LIN {X 0,Y 573.271,Z 613.194,A -85,B 0,C 180,E1 -2290.528,E2 -2290.528} C_VEL
LIN {X 0,Y 573.246,Z 613.204,A -85,B 0,C 180,E1 -2293.669,E2 -2293.669} C_VEL
LIN {X 0,Y 573.242,Z 613.198,A -85,B 0,C 180,E1 -2296.641,E2 -2296.641} C_VEL
LIN {X 0,Y 573.276,Z 613.202,A -85,B 0,C 180,E1 -2299.478,E2 -2299.478} C_VEL
LIN {X 0,Y 573.238,Z 613.198,A -85,B 0,C 180,E1 -2302.193,E2 -2302.193} C_VEL
LIN {X 0,Y 573.271,Z 613.195,A -85,B 0,C 180,E1 -2304.817,E2 -2304.817} C_VEL
LIN {X 0,Y 573.259,Z 613.2,A -85,B 0,C 180,E1 -2307.355,E2 -2307.355} C_VEL
LIN {X 0,Y 573.252,Z 613.206,A -85,B 0,C 180,E1 -2309.824,E2 -2309.824} C_VEL
LIN {X 0,Y 573.291,Z 613.195,A -85,B 0,C 180,E1 -2312.235,E2 -2312.235} C_VEL
LIN {X 0,Y 573.277,Z 613.196,A -85,B 0,C 180,E1 -2315.366,E2 -2315.366} C_VEL
LIN {X 0,Y 573.232,Z 613.202,A -85,B 0,C 180,E1 -2318.42,E2 -2318.42} C_VEL
LIN {X 0,Y 573.281,Z 613.193,A -85,B 0,C 180,E1 -2320.728,E2 -2320.728} C_VEL
LIN {X 0,Y 573.261,Z 613.2,A -85,B 0,C 180,E1 -2323.622,E2 -2323.622} C_VEL
LIN {X 0,Y 573.275,Z 613.2,A -85,B 0,C 180,E1 -2325.807,E2 -2325.807} C_VEL
LIN {X 0,Y 573.265,Z 613.197,A -85,B 0,C 180,E1 -2328.745,E2 -2328.745} C_VEL
LIN {X 0,Y 573.287,Z 613.193,A -85,B 0,C 180,E1 -2331.541,E2 -2331.541} C_VEL
LIN {X 0,Y 573.287,Z 613.2,A -85,B 0,C 180,E1 -2334.372,E2 -2334.372} C_VEL
LIN {X 0,Y 573.309,Z 613.19,A -85,B 0,C 180,E1 -2337.19,E2 -2337.19} C_VEL
LIN {X 0,Y 573.324,Z 613.193,A -85,B 0,C 180,E1 -2340,E2 -2340} C_VEL
LIN {X 0,Y 573.303,Z 613.194,A -85,B 0,C 180,E1 -2342.811,E2 -2342.811} C_VEL
LIN {X 0,Y 573.293,Z 613.191,A -85,B 0,C 180,E1 -2345.628,E2 -2345.628} C_VEL
LIN {X 0,Y 573.286,Z 613.203,A -85,B 0,C 180,E1 -2348.46,E2 -2348.46} C_VEL
LIN {X 0,Y 573.275,Z 613.194,A -85,B 0,C 180,E1 -2351.312,E2 -2351.312} C_VEL
LIN {X 0,Y 573.284,Z 613.2,A -85,B 0,C 180,E1 -2354.424,E2 -2354.424} C_VEL
LIN {X 0,Y 573.261,Z 613.199,A -85,B 0,C 180,E1 -2357.112,E2 -2357.112} C_VEL
LIN {X 0,Y 573.244,Z 613.198,A -85,B 0,C 180,E1 -2360.077,E2 -2360.077} C_VEL
LIN {X 0,Y 573.234,Z 613.203,A -85,B 0,C 180,E1 -2362.338,E2 -2362.338} C_VEL
LIN {X 0,Y 573.248,Z 613.2,A -85,B 0,C 180,E1 -2364.387,E2 -2364.387} C_VEL
LIN {X 0,Y 572.619,Z 613.286,A -85,B 0,C 180,E1 -2364.973,E2 -2364.973} C_VEL
LIN {X 0,Y 569.76,Z 613.642,A -85,B 0,C 180,E1 -2365.924,E2 -2365.924} C_VEL
LIN {X 0,Y 567.315,Z 613.945,A -85,B 0,C 180,E1 -2366.689,E2 -2366.689} C_VEL
LIN {X 0,Y 566.258,Z 614.07,A -85,B 0,C 180,E1 -2367.281,E2 -2367.281} C_VEL
LIN {X 0,Y 566.17,Z 614.079,A -85,B 0,C 180,E1 -2367.481,E2 -2367.481} C_VEL
LIN {X 0,Y 566.199,Z 614.073,A -85,B 0,C 180,E1 -2369.769,E2 -2369.769} C_VEL
LIN {X 0,Y 566.206,Z 614.077,A -85,B 0,C 180,E1 -2372.43,E2 -2372.43} C_VEL
LIN {X 0,Y 566.18,Z 614.088,A -85,B 0,C 180,E1 -2374.989,E2 -2374.989} C_VEL
LIN {X 0,Y 566.197,Z 614.08,A -85,B 0,C 180,E1 -2377.461,E2 -2377.461} C_VEL
LIN {X 0,Y 566.209,Z 614.073,A -85,B 0,C 180,E1 -2380.199,E2 -2380.199} C_VEL
LIN {X 0,Y 566.184,Z 614.087,A -85,B 0,C 180,E1 -2383.056,E2 -2383.056} C_VEL
LIN {X 0,Y 566.159,Z 614.081,A -85,B 0,C 180,E1 -2386.053,E2 -2386.053} C_VEL
LIN {X 0,Y 566.167,Z 614.084,A -85,B 0,C 180,E1 -2388.86,E2 -2388.86} C_VEL
LIN {X 0,Y 566.206,Z 614.084,A -85,B 0,C 180,E1 -2391.443,E2 -2391.443} C_VEL
LIN {X 0,Y 566.148,Z 614.082,A -85,B 0,C 180,E1 -2394.307,E2 -2394.307} C_VEL
LIN {X 0,Y 566.198,Z 614.078,A -85,B 0,C 180,E1 -2396.896,E2 -2396.896} C_VEL
LIN {X 0,Y 566.169,Z 614.089,A -85,B 0,C 180,E1 -2399.407,E2 -2399.407} C_VEL
LIN {X 0,Y 566.174,Z 614.086,A -85,B 0,C 180,E1 -2401.855,E2 -2401.855} C_VEL
LIN {X 0,Y 566.21,Z 614.214,A -85,B 0,C 180,E1 -2404.103,E2 -2404.103} C_VEL
LIN {X 0,Y 566.783,Z 618.685,A -85,B 0,C 180,E1 -2404.849,E2 -2404.849} C_VEL
LIN {X 0,Y 566.52,Z 638.155,A -85,B 0,C 180,E1 -2407.959,E2 -2407.959} C_VEL
LIN {X 0,Y 566.539,Z 638.91,A -85,B 0,C 180,E1 -2408.08,E2 -2408.08} C_VEL
LIN {X 0,Y 567.797,Z 645.92,A -85,B 0,C 180,E1 -2408.214,E2 -2408.214} C_VEL
LIN {X 0,Y 567.426,Z 775.387,A -85,B 0,C 180,E1 -2409.89,E2 -2409.89} C_VEL
LIN {X 0,Y 567.273,Z 789.85,A -85,B 0,C 180,E1 -2410.224,E2 -2410.224} C_VEL
LIN {X 0,Y 567.158,Z 803.531,A -85,B 0,C 180,E1 -2410.689,E2 -2410.689} C_VEL
LIN {X 0,Y 566.982,Z 816.893,A -85,B 0,C 180,E1 -2411.293,E2 -2411.293} C_VEL
LIN {X 0,Y 566.77,Z 829.75,A -85,B 0,C 180,E1 -2412.034,E2 -2412.034} C_VEL
LIN {X 0,Y 566.592,Z 841.641,A -85,B 0,C 180,E1 -2412.884,E2 -2412.884} C_VEL
LIN {X 0,Y 566.402,Z 852.078,A -85,B 0,C 180,E1 -2413.789,E2 -2413.789} C_VEL
LIN {X 0,Y 566.259,Z 862.634,A -85,B 0,C 180,E1 -2414.892,E2 -2414.892} C_VEL
LIN {X 0,Y 566.111,Z 871.296,A -85,B 0,C 180,E1 -2415.991,E2 -2415.991} C_VEL
LIN {X 0,Y 566.028,Z 879.528,A -85,B 0,C 180,E1 -2417.268,E2 -2417.268} C_VEL
LIN {X 0,Y 565.938,Z 886.128,A -85,B 0,C 180,E1 -2418.539,E2 -2418.539} C_VEL
LIN {X 0,Y 565.917,Z 890.69,A -85,B 0,C 180,E1 -2419.626,E2 -2419.626} C_VEL
LIN {X 0,Y 565.877,Z 894.258,A -85,B 0,C 180,E1 -2420.709,E2 -2420.709} C_VEL
LIN {X 0,Y 565.882,Z 897.734,A -85,B 0,C 180,E1 -2422.148,E2 -2422.148} C_VEL
LIN {X 0,Y 565.899,Z 899.79,A -85,B 0,C 180,E1 -2423.583,E2 -2423.583} C_VEL
LIN {X 0,Y 565.844,Z 900.498,A -85,B 0,C 180,E1 -2425.012,E2 -2425.012} C_VEL
LIN {X 0,Y 565.885,Z 899.863,A -85,B 0,C 180,E1 -2426.44,E2 -2426.44} C_VEL
LIN {X 0,Y 565.839,Z 897.888,A -85,B 0,C 180,E1 -2427.865,E2 -2427.865} C_VEL
LIN {X 0,Y 565.848,Z 894.533,A -85,B 0,C 180,E1 -2429.288,E2 -2429.288} C_VEL
LIN {X 0,Y 565.89,Z 889.709,A -85,B 0,C 180,E1 -2430.712,E2 -2430.712} C_VEL
LIN {X 0,Y 566.002,Z 885.069,A -85,B 0,C 180,E1 -2431.779,E2 -2431.779} C_VEL
LIN {X 0,Y 566.061,Z 878.343,A -85,B 0,C 180,E1 -2433.025,E2 -2433.025} C_VEL
LIN {X 0,Y 566.16,Z 870.011,A -85,B 0,C 180,E1 -2434.271,E2 -2434.271} C_VEL
LIN {X 0,Y 566.241,Z 861.352,A -85,B 0,C 180,E1 -2435.341,E2 -2435.341} C_VEL
LIN {X 0,Y 566.433,Z 850.893,A -85,B 0,C 180,E1 -2436.412,E2 -2436.412} C_VEL
LIN {X 0,Y 566.652,Z 839.212,A -85,B 0,C 180,E1 -2437.393,E2 -2437.393} C_VEL
LIN {X 0,Y 566.807,Z 827.519,A -85,B 0,C 180,E1 -2438.198,E2 -2438.198} C_VEL
LIN {X 0,Y 566.977,Z 814.646,A -85,B 0,C 180,E1 -2438.914,E2 -2438.914} C_VEL
LIN {X 0,Y 567.184,Z 801.171,A -85,B 0,C 180,E1 -2439.495,E2 -2439.495} C_VEL
LIN {X 0,Y 567.297,Z 787.032,A -85,B 0,C 180,E1 -2439.943,E2 -2439.943} C_VEL
LIN {X 0,Y 567.415,Z 773.297,A -85,B 0,C 180,E1 -2440.234,E2 -2440.234} C_VEL
LIN {X 0,Y 567.787,Z 645.918,A -85,B 0,C 180,E1 -2441.877,E2 -2441.877} C_VEL
LIN {X 0,Y 566.495,Z 638.792,A -85,B 0,C 180,E1 -2442.03,E2 -2442.03} C_VEL
LIN {X 0,Y 566.712,Z 622.116,A -85,B 0,C 180,E1 -2444.69,E2 -2444.69} C_VEL
LIN {X 0,Y 566.544,Z 616.194,A -85,B 0,C 180,E1 -2445.653,E2 -2445.653} C_VEL
LIN {X 0,Y 566.179,Z 614.087,A -85,B 0,C 180,E1 -2446.033,E2 -2446.033} C_VEL
LIN {X 0,Y 566.172,Z 614.088,A -85,B 0,C 180,E1 -2448.829,E2 -2448.829} C_VEL
LIN {X 0,Y 566.211,Z 614.076,A -85,B 0,C 180,E1 -2451.419,E2 -2451.419} C_VEL
LIN {X 0,Y 566.154,Z 614.085,A -85,B 0,C 180,E1 -2454.183,E2 -2454.183} C_VEL
LIN {X 0,Y 566.165,Z 614.09,A -85,B 0,C 180,E1 -2456.649,E2 -2456.649} C_VEL
LIN {X 0,Y 566.159,Z 614.081,A -85,B 0,C 180,E1 -2459.771,E2 -2459.771} C_VEL
LIN {X 0,Y 566.18,Z 614.082,A -85,B 0,C 180,E1 -2462.425,E2 -2462.425} C_VEL
LIN {X 0,Y 566.165,Z 614.089,A -85,B 0,C 180,E1 -2464.986,E2 -2464.986} C_VEL
LIN {X 0,Y 566.188,Z 614.079,A -85,B 0,C 180,E1 -2467.462,E2 -2467.462} C_VEL
LIN {X 0,Y 566.169,Z 614.077,A -85,B 0,C 180,E1 -2470.203,E2 -2470.203} C_VEL
LIN {X 0,Y 566.181,Z 614.087,A -85,B 0,C 180,E1 -2473.056,E2 -2473.056} C_VEL
LIN {X 0,Y 566.158,Z 614.081,A -85,B 0,C 180,E1 -2476.053,E2 -2476.053} C_VEL
LIN {X 0,Y 566.154,Z 614.087,A -85,B 0,C 180,E1 -2478.858,E2 -2478.858} C_VEL
LIN {X 0,Y 566.201,Z 614.078,A -85,B 0,C 180,E1 -2481.444,E2 -2481.444} C_VEL
LIN {X 0,Y 566.145,Z 614.08,A -85,B 0,C 180,E1 -2484.306,E2 -2484.306} C_VEL
LIN {X 0,Y 566.2,Z 614.08,A -85,B 0,C 180,E1 -2486.896,E2 -2486.896} C_VEL
LIN {X 0,Y 566.171,Z 614.086,A -85,B 0,C 180,E1 -2489.406,E2 -2489.406} C_VEL
LIN {X 0,Y 566.191,Z 614.079,A -85,B 0,C 180,E1 -2491.856,E2 -2491.856} C_VEL
LIN {X 0,Y 566.185,Z 614.077,A -85,B 0,C 180,E1 -2494.249,E2 -2494.249} C_VEL
LIN {X 0,Y 566.169,Z 614.078,A -85,B 0,C 180,E1 -2496.72,E2 -2496.72} C_VEL
LIN {X 0,Y 566.208,Z 614.081,A -85,B 0,C 180,E1 -2499.662,E2 -2499.662} C_VEL
LIN {X 0,Y 566.197,Z 614.073,A -85,B 0,C 180,E1 -2502.668,E2 -2502.668} C_VEL
LIN {X 0,Y 566.237,Z 614.08,A -85,B 0,C 180,E1 -2505.627,E2 -2505.627} C_VEL
LIN {X 0,Y 566.239,Z 614.069,A -85,B 0,C 180,E1 -2508.675,E2 -2508.675} C_VEL
LIN {X 0,Y 566.226,Z 614.077,A -85,B 0,C 180,E1 -2511.434,E2 -2511.434} C_VEL
LIN {X 0,Y 566.25,Z 614.07,A -85,B 0,C 180,E1 -2514.301,E2 -2514.301} C_VEL
LIN {X 0,Y 566.283,Z 614.074,A -85,B 0,C 180,E1 -2517.866,E2 -2517.866} C_VEL
LIN {X 0,Y 566.302,Z 614.062,A -85,B 0,C 180,E1 -2520.711,E2 -2520.711} C_VEL
LIN {X 0,Y 566.273,Z 614.066,A -85,B 0,C 180,E1 -2522.845,E2 -2522.845} C_VEL
LIN {X 0,Y 566.256,Z 614.075,A -85,B 0,C 180,E1 -2525.698,E2 -2525.698} C_VEL
LIN {X 0,Y 566.23,Z 614.073,A -85,B 0,C 180,E1 -2528.566,E2 -2528.566} C_VEL
LIN {X 0,Y 566.245,Z 614.071,A -85,B 0,C 180,E1 -2531.454,E2 -2531.454} C_VEL
LIN {X 0,Y 566.238,Z 614.073,A -85,B 0,C 180,E1 -2534.506,E2 -2534.506} C_VEL
LIN {X 0,Y 566.203,Z 614.075,A -85,B 0,C 180,E1 -2537.331,E2 -2537.331} C_VEL
LIN {X 0,Y 566.217,Z 614.08,A -85,B 0,C 180,E1 -2540.337,E2 -2540.337} C_VEL
LIN {X 0,Y 566.172,Z 614.078,A -85,B 0,C 180,E1 -2543.281,E2 -2543.281} C_VEL
LIN {X 0,Y 566.215,Z 614.076,A -85,B 0,C 180,E1 -2545.749,E2 -2545.749} C_VEL
LIN {X 0,Y 566.205,Z 614.084,A -85,B 0,C 180,E1 -2548.202,E2 -2548.202} C_VEL
LIN {X 0,Y 566.197,Z 614.076,A -85,B 0,C 180,E1 -2551.077,E2 -2551.077} C_VEL
LIN {X 0,Y 566.215,Z 614.075,A -85,B 0,C 180,E1 -2553.734,E2 -2553.734} C_VEL
LIN {X 0,Y 566.203,Z 614.083,A -85,B 0,C 180,E1 -2556.57,E2 -2556.57} C_VEL
LIN {X 0,Y 566.224,Z 614.072,A -85,B 0,C 180,E1 -2559.273,E2 -2559.273} C_VEL
LIN {X 0,Y 566.194,Z 614.08,A -85,B 0,C 180,E1 -2562.089,E2 -2562.089} C_VEL
LIN {X 0,Y 566.175,Z 614.081,A -85,B 0,C 180,E1 -2565.036,E2 -2565.036} C_VEL
LIN {X 0,Y 566.221,Z 614.076,A -85,B 0,C 180,E1 -2568.136,E2 -2568.136} C_VEL
LIN {X 0,Y 566.218,Z 614.083,A -85,B 0,C 180,E1 -2570.726,E2 -2570.726} C_VEL
LIN {X 0,Y 566.22,Z 614.074,A -85,B 0,C 180,E1 -2573.783,E2 -2573.783} C_VEL
LIN {X 0,Y 566.215,Z 614.077,A -85,B 0,C 180,E1 -2576.266,E2 -2576.266} C_VEL
LIN {X 0,Y 566.202,Z 614.084,A -85,B 0,C 180,E1 -2578.922,E2 -2578.922} C_VEL
LIN {X 0,Y 566.214,Z 614.075,A -85,B 0,C 180,E1 -2581.857,E2 -2581.857} C_VEL
LIN {X 0,Y 566.22,Z 614.081,A -85,B 0,C 180,E1 -2584.644,E2 -2584.644} C_VEL
LIN {X 0,Y 566.24,Z 614.207,A -85,B 0,C 180,E1 -2584.792,E2 -2584.792} C_VEL
LIN {X 0,Y 567.536,Z 620.359,A -85,B 0,C 180,E1 -2585.685,E2 -2585.685} C_VEL
LIN {X 0,Y 567.212,Z 640.232,A -85,B 0,C 180,E1 -2588.323,E2 -2588.323} C_VEL
LIN {X 0,Y 566.892,Z 662.255,A -85,B 0,C 180,E1 -2591.196,E2 -2591.196} C_VEL
LIN {X 0,Y 566.687,Z 676.414,A -85,B 0,C 180,E1 -2593.018,E2 -2593.018} C_VEL
LIN {X 0,Y 567.814,Z 683.83,A -85,B 0,C 180,E1 -2593.155,E2 -2593.155} C_VEL
LIN {X 0,Y 567.43,Z 814.879,A -85,B 0,C 180,E1 -2594.855,E2 -2594.855} C_VEL
LIN {X 0,Y 567.273,Z 829.536,A -85,B 0,C 180,E1 -2595.2,E2 -2595.2} C_VEL
LIN {X 0,Y 567.102,Z 843.837,A -85,B 0,C 180,E1 -2595.695,E2 -2595.695} C_VEL
LIN {X 0,Y 566.964,Z 856.64,A -85,B 0,C 180,E1 -2596.286,E2 -2596.286} C_VEL
LIN {X 0,Y 566.787,Z 869.098,A -85,B 0,C 180,E1 -2597.012,E2 -2597.012} C_VEL
LIN {X 0,Y 566.576,Z 880.478,A -85,B 0,C 180,E1 -2597.826,E2 -2597.826} C_VEL
LIN {X 0,Y 566.452,Z 891.045,A -85,B 0,C 180,E1 -2598.742,E2 -2598.742} C_VEL
LIN {X 0,Y 566.247,Z 901.333,A -85,B 0,C 180,E1 -2599.813,E2 -2599.813} C_VEL
LIN {X 0,Y 566.153,Z 909.911,A -85,B 0,C 180,E1 -2600.893,E2 -2600.893} C_VEL
LIN {X 0,Y 566.059,Z 918.115,A -85,B 0,C 180,E1 -2602.15,E2 -2602.15} C_VEL
LIN {X 0,Y 565.966,Z 924.801,A -85,B 0,C 180,E1 -2603.422,E2 -2603.422} C_VEL
LIN {X 0,Y 565.927,Z 929.961,A -85,B 0,C 180,E1 -2604.656,E2 -2604.656} C_VEL
LIN {X 0,Y 565.957,Z 933.443,A -85,B 0,C 180,E1 -2605.727,E2 -2605.727} C_VEL
LIN {X 0,Y 565.874,Z 936.831,A -85,B 0,C 180,E1 -2607.152,E2 -2607.152} C_VEL
LIN {X 0,Y 565.84,Z 938.832,A -85,B 0,C 180,E1 -2608.576,E2 -2608.576} C_VEL
LIN {X 0,Y 565.837,Z 939.5,A -85,B 0,C 180,E1 -2610,E2 -2610} C_VEL
LIN {X 0,Y 565.84,Z 938.833,A -85,B 0,C 180,E1 -2611.423,E2 -2611.423} C_VEL
LIN {X 0,Y 565.874,Z 936.833,A -85,B 0,C 180,E1 -2612.847,E2 -2612.847} C_VEL
LIN {X 0,Y 565.956,Z 933.445,A -85,B 0,C 180,E1 -2614.273,E2 -2614.273} C_VEL
LIN {X 0,Y 565.988,Z 928.568,A -85,B 0,C 180,E1 -2615.701,E2 -2615.701} C_VEL
LIN {X 0,Y 565.992,Z 924.045,A -85,B 0,C 180,E1 -2616.739,E2 -2616.739} C_VEL
LIN {X 0,Y 566.047,Z 917.038,A -85,B 0,C 180,E1 -2618.029,E2 -2618.029} C_VEL
LIN {X 0,Y 566.177,Z 908.559,A -85,B 0,C 180,E1 -2619.286,E2 -2619.286} C_VEL
LIN {X 0,Y 566.294,Z 899.708,A -85,B 0,C 180,E1 -2620.367,E2 -2620.367} C_VEL
LIN {X 0,Y 566.485,Z 888.991,A -85,B 0,C 180,E1 -2621.449,E2 -2621.449} C_VEL
LIN {X 0,Y 566.629,Z 878.143,A -85,B 0,C 180,E1 -2622.354,E2 -2622.354} C_VEL
LIN {X 0,Y 566.8,Z 866.259,A -85,B 0,C 180,E1 -2623.17,E2 -2623.17} C_VEL
LIN {X 0,Y 567.02,Z 853.096,A -85,B 0,C 180,E1 -2623.895,E2 -2623.895} C_VEL
LIN {X 0,Y 567.192,Z 840.055,A -85,B 0,C 180,E1 -2624.453,E2 -2624.453} C_VEL
LIN {X 0,Y 567.324,Z 826.235,A -85,B 0,C 180,E1 -2624.892,E2 -2624.892} C_VEL
LIN {X 0,Y 567.455,Z 812.133,A -85,B 0,C 180,E1 -2625.19,E2 -2625.19} C_VEL
LIN {X 0,Y 567.765,Z 682.287,A -85,B 0,C 180,E1 -2626.867,E2 -2626.867} C_VEL
LIN {X 0,Y 566.685,Z 676.417,A -85,B 0,C 180,E1 -2626.981,E2 -2626.981} C_VEL
LIN {X 0,Y 566.979,Z 655.178,A -85,B 0,C 180,E1 -2629.723,E2 -2629.723} C_VEL
LIN {X 0,Y 567.374,Z 631.917,A -85,B 0,C 180,E1 -2632.774,E2 -2632.774} C_VEL
LIN {X 0,Y 567.535,Z 620.36,A -85,B 0,C 180,E1 -2634.315,E2 -2634.315} C_VEL
LIN {X 0,Y 566.224,Z 614.081,A -85,B 0,C 180,E1 -2635.257,E2 -2635.257} C_VEL
LIN {X 0,Y 566.231,Z 614.074,A -85,B 0,C 180,E1 -2638.142,E2 -2638.142} C_VEL
LIN {X 0,Y 566.201,Z 614.084,A -85,B 0,C 180,E1 -2641.078,E2 -2641.078} C_VEL
LIN {X 0,Y 566.214,Z 614.077,A -85,B 0,C 180,E1 -2643.734,E2 -2643.734} C_VEL
LIN {X 0,Y 566.218,Z 614.074,A -85,B 0,C 180,E1 -2646.569,E2 -2646.569} C_VEL
LIN {X 0,Y 566.214,Z 614.078,A -85,B 0,C 180,E1 -2649.686,E2 -2649.686} C_VEL
LIN {X 0,Y 566.215,Z 614.075,A -85,B 0,C 180,E1 -2652.087,E2 -2652.087} C_VEL
LIN {X 0,Y 566.174,Z 614.081,A -85,B 0,C 180,E1 -2655.036,E2 -2655.036} C_VEL
LIN {X 0,Y 566.22,Z 614.074,A -85,B 0,C 180,E1 -2658.136,E2 -2658.136} C_VEL
LIN {X 0,Y 566.224,Z 614.073,A -85,B 0,C 180,E1 -2660.727,E2 -2660.727} C_VEL
LIN {X 0,Y 566.22,Z 614.081,A -85,B 0,C 180,E1 -2663.783,E2 -2663.783} C_VEL
LIN {X 0,Y 566.214,Z 614.075,A -85,B 0,C 180,E1 -2666.266,E2 -2666.266} C_VEL
LIN {X 0,Y 566.201,Z 614.071,A -85,B 0,C 180,E1 -2668.922,E2 -2668.922} C_VEL
LIN {X 0,Y 566.231,Z 614.081,A -85,B 0,C 180,E1 -2671.858,E2 -2671.858} C_VEL
LIN {X 0,Y 566.215,Z 614.077,A -85,B 0,C 180,E1 -2674.251,E2 -2674.251} C_VEL
LIN {X 0,Y 566.193,Z 614.076,A -85,B 0,C 180,E1 -2676.714,E2 -2676.714} C_VEL
LIN {X 0,Y 566.216,Z 614.079,A -85,B 0,C 180,E1 -2679.663,E2 -2679.663} C_VEL
LIN {X 0,Y 566.206,Z 614.076,A -85,B 0,C 180,E1 -2682.669,E2 -2682.669} C_VEL
LIN {X 0,Y 566.236,Z 614.074,A -85,B 0,C 180,E1 -2685.627,E2 -2685.627} C_VEL
LIN {X 0,Y 566.237,Z 614.073,A -85,B 0,C 180,E1 -2688.675,E2 -2688.675} C_VEL
LIN {X 0,Y 566.23,Z 614.071,A -85,B 0,C 180,E1 -2691.434,E2 -2691.434} C_VEL
LIN {X 0,Y 566.256,Z 614.077,A -85,B 0,C 180,E1 -2694.302,E2 -2694.302} C_VEL
LIN {X 0,Y 566.282,Z 614.069,A -85,B 0,C 180,E1 -2697.866,E2 -2697.866} C_VEL
LIN {X 0,Y 566.3,Z 614.067,A -85,B 0,C 180,E1 -2700.711,E2 -2700.711} C_VEL
LIN {X 0,Y 566.27,Z 614.07,A -85,B 0,C 180,E1 -2702.846,E2 -2702.846} C_VEL
LIN {X 0,Y 566.262,Z 614.067,A -85,B 0,C 180,E1 -2705.698,E2 -2705.698} C_VEL
LIN {X 0,Y 566.229,Z 614.081,A -85,B 0,C 180,E1 -2708.566,E2 -2708.566} C_VEL
LIN {X 0,Y 566.245,Z 614.07,A -85,B 0,C 180,E1 -2711.455,E2 -2711.455} C_VEL
LIN {X 0,Y 566.237,Z 614.08,A -85,B 0,C 180,E1 -2714.507,E2 -2714.507} C_VEL
LIN {X 0,Y 566.201,Z 614.077,A -85,B 0,C 180,E1 -2717.332,E2 -2717.332} C_VEL
LIN {X 0,Y 566.21,Z 614.077,A -85,B 0,C 180,E1 -2720.338,E2 -2720.338} C_VEL
LIN {X 0,Y 566.17,Z 614.081,A -85,B 0,C 180,E1 -2723.281,E2 -2723.281} C_VEL
LIN {X 0,Y 566.206,Z 614.075,A -85,B 0,C 180,E1 -2725.75,E2 -2725.75} C_VEL
LIN {X 0,Y 566.17,Z 614.079,A -85,B 0,C 180,E1 -2727.481,E2 -2727.481} C_VEL
LIN {X 0,Y 565.499,Z 614.162,A -85,B 0,C 180,E1 -2728.075,E2 -2728.075} C_VEL
LIN {X 0,Y 562.646,Z 614.523,A -85,B 0,C 180,E1 -2729.039,E2 -2729.039} C_VEL
LIN {X 0,Y 560.242,Z 614.818,A -85,B 0,C 180,E1 -2729.815,E2 -2729.815} C_VEL
LIN {X 0,Y 559.217,Z 614.945,A -85,B 0,C 180,E1 -2730.414,E2 -2730.414} C_VEL
LIN {X 0,Y 559.137,Z 614.957,A -85,B 0,C 180,E1 -2730.616,E2 -2730.616} C_VEL
LIN {X 0,Y 559.154,Z 614.96,A -85,B 0,C 180,E1 -2732.716,E2 -2732.716} C_VEL
LIN {X 0,Y 559.129,Z 614.961,A -85,B 0,C 180,E1 -2735.324,E2 -2735.324} C_VEL
LIN {X 0,Y 559.131,Z 614.956,A -85,B 0,C 180,E1 -2738.018,E2 -2738.018} C_VEL
LIN {X 0,Y 559.155,Z 614.957,A -85,B 0,C 180,E1 -2740.813,E2 -2740.813} C_VEL
LIN {X 0,Y 559.111,Z 614.961,A -85,B 0,C 180,E1 -2743.737,E2 -2743.737} C_VEL
LIN {X 0,Y 559.11,Z 614.959,A -85,B 0,C 180,E1 -2746.263,E2 -2746.263} C_VEL
LIN {X 0,Y 559.155,Z 614.963,A -85,B 0,C 180,E1 -2749.187,E2 -2749.187} C_VEL
LIN {X 0,Y 559.131,Z 614.958,A -85,B 0,C 180,E1 -2751.982,E2 -2751.982} C_VEL
LIN {X 0,Y 559.127,Z 614.958,A -85,B 0,C 180,E1 -2754.789,E2 -2754.789} C_VEL
LIN {X 0,Y 559.152,Z 614.96,A -85,B 0,C 180,E1 -2757.366,E2 -2757.366} C_VEL
LIN {X 0,Y 559.12,Z 614.96,A -85,B 0,C 180,E1 -2760.149,E2 -2760.149} C_VEL
LIN {X 0,Y 559.114,Z 614.967,A -85,B 0,C 180,E1 -2763.185,E2 -2763.185} C_VEL
LIN {X 0,Y 559.163,Z 614.979,A -85,B 0,C 180,E1 -2763.952,E2 -2763.952} C_VEL
LIN {X 0,Y 559.795,Z 619.574,A -85,B 0,C 180,E1 -2764.732,E2 -2764.732} C_VEL
LIN {X 0,Y 559.524,Z 637.72,A -85,B 0,C 180,E1 -2767.669,E2 -2767.669} C_VEL
LIN {X 0,Y 559.518,Z 638.927,A -85,B 0,C 180,E1 -2767.863,E2 -2767.863} C_VEL
LIN {X 0,Y 561.012,Z 646.832,A -85,B 0,C 180,E1 -2768.016,E2 -2768.016} C_VEL
LIN {X 0,Y 560.608,Z 774.759,A -85,B 0,C 180,E1 -2769.69,E2 -2769.69} C_VEL
LIN {X 0,Y 560.462,Z 788.934,A -85,B 0,C 180,E1 -2770.012,E2 -2770.012} C_VEL
LIN {X 0,Y 560.274,Z 803.153,A -85,B 0,C 180,E1 -2770.493,E2 -2770.493} C_VEL
LIN {X 0,Y 560.077,Z 815.624,A -85,B 0,C 180,E1 -2771.053,E2 -2771.053} C_VEL
LIN {X 0,Y 559.86,Z 827.273,A -85,B 0,C 180,E1 -2771.71,E2 -2771.71} C_VEL
LIN {X 0,Y 559.653,Z 839.346,A -85,B 0,C 180,E1 -2772.55,E2 -2772.55} C_VEL
LIN {X 0,Y 559.469,Z 849.397,A -85,B 0,C 180,E1 -2773.394,E2 -2773.394} C_VEL
LIN {X 0,Y 559.287,Z 858.744,A -85,B 0,C 180,E1 -2774.326,E2 -2774.326} C_VEL
LIN {X 0,Y 559.123,Z 868.85,A -85,B 0,C 180,E1 -2775.545,E2 -2775.545} C_VEL
LIN {X 0,Y 558.994,Z 876.943,A -85,B 0,C 180,E1 -2776.735,E2 -2776.735} C_VEL
LIN {X 0,Y 558.888,Z 884.071,A -85,B 0,C 180,E1 -2778.025,E2 -2778.025} C_VEL
LIN {X 0,Y 558.859,Z 889.002,A -85,B 0,C 180,E1 -2779.127,E2 -2779.127} C_VEL
LIN {X 0,Y 558.793,Z 894.072,A -85,B 0,C 180,E1 -2780.59,E2 -2780.59} C_VEL
LIN {X 0,Y 558.801,Z 897.609,A -85,B 0,C 180,E1 -2782.048,E2 -2782.048} C_VEL
LIN {X 0,Y 558.827,Z 899.723,A -85,B 0,C 180,E1 -2783.501,E2 -2783.501} C_VEL
LIN {X 0,Y 558.759,Z 900.485,A -85,B 0,C 180,E1 -2784.949,E2 -2784.949} C_VEL
LIN {X 0,Y 558.797,Z 899.919,A -85,B 0,C 180,E1 -2786.395,E2 -2786.395} C_VEL
LIN {X 0,Y 558.744,Z 898.012,A -85,B 0,C 180,E1 -2787.838,E2 -2787.838} C_VEL
LIN {X 0,Y 558.749,Z 894.718,A -85,B 0,C 180,E1 -2789.279,E2 -2789.279} C_VEL
LIN {X 0,Y 558.796,Z 889.957,A -85,B 0,C 180,E1 -2790.721,E2 -2790.721} C_VEL
LIN {X 0,Y 558.91,Z 885.373,A -85,B 0,C 180,E1 -2791.802,E2 -2791.802} C_VEL
LIN {X 0,Y 559.008,Z 878.725,A -85,B 0,C 180,E1 -2793.063,E2 -2793.063} C_VEL
LIN {X 0,Y 559.12,Z 870.481,A -85,B 0,C 180,E1 -2794.325,E2 -2794.325} C_VEL
LIN {X 0,Y 559.21,Z 861.916,A -85,B 0,C 180,E1 -2795.409,E2 -2795.409} C_VEL
LIN {X 0,Y 559.411,Z 851.567,A -85,B 0,C 180,E1 -2796.492,E2 -2796.492} C_VEL
LIN {X 0,Y 559.659,Z 840.024,A -85,B 0,C 180,E1 -2797.486,E2 -2797.486} C_VEL
LIN {X 0,Y 559.857,Z 828.502,A -85,B 0,C 180,E1 -2798.3,E2 -2798.3} C_VEL
LIN {X 0,Y 560.043,Z 815.863,A -85,B 0,C 180,E1 -2799.025,E2 -2799.025} C_VEL
LIN {X 0,Y 560.291,Z 802.768,A -85,B 0,C 180,E1 -2799.613,E2 -2799.613} C_VEL
LIN {X 0,Y 560.472,Z 788.582,A -85,B 0,C 180,E1 -2800.088,E2 -2800.088} C_VEL
LIN {X 0,Y 560.571,Z 774.462,A -85,B 0,C 180,E1 -2800.406,E2 -2800.406} C_VEL
LIN {X 0,Y 560.974,Z 646.407,A -85,B 0,C 180,E1 -2802.081,E2 -2802.081} C_VEL
LIN {X 0,Y 559.505,Z 638.834,A -85,B 0,C 180,E1 -2802.243,E2 -2802.243} C_VEL
LIN {X 0,Y 559.794,Z 621.074,A -85,B 0,C 180,E1 -2805.113,E2 -2805.113} C_VEL
LIN {X 0,Y 559.465,Z 616.617,A -85,B 0,C 180,E1 -2805.856,E2 -2805.856} C_VEL
LIN {X 0,Y 559.136,Z 614.965,A -85,B 0,C 180,E1 -2806.147,E2 -2806.147} C_VEL
LIN {X 0,Y 559.139,Z 614.961,A -85,B 0,C 180,E1 -2809.075,E2 -2809.075} C_VEL
LIN {X 0,Y 559.155,Z 614.955,A -85,B 0,C 180,E1 -2811.548,E2 -2811.548} C_VEL
LIN {X 0,Y 559.092,Z 614.969,A -85,B 0,C 180,E1 -2814.508,E2 -2814.508} C_VEL
LIN {X 0,Y 559.112,Z 614.967,A -85,B 0,C 180,E1 -2816.905,E2 -2816.905} C_VEL
LIN {X 0,Y 559.109,Z 614.959,A -85,B 0,C 180,E1 -2819.849,E2 -2819.849} C_VEL
LIN {X 0,Y 559.138,Z 614.964,A -85,B 0,C 180,E1 -2822.717,E2 -2822.717} C_VEL
LIN {X 0,Y 559.117,Z 614.961,A -85,B 0,C 180,E1 -2825.325,E2 -2825.325} C_VEL
LIN {X 0,Y 559.125,Z 614.957,A -85,B 0,C 180,E1 -2828.018,E2 -2828.018} C_VEL
LIN {X 0,Y 559.105,Z 614.964,A -85,B 0,C 180,E1 -2830.817,E2 -2830.817} C_VEL
LIN {X 0,Y 559.11,Z 614.959,A -85,B 0,C 180,E1 -2833.737,E2 -2833.737} C_VEL
LIN {X 0,Y 559.109,Z 614.959,A -85,B 0,C 180,E1 -2836.262,E2 -2836.262} C_VEL
LIN {X 0,Y 559.127,Z 614.966,A -85,B 0,C 180,E1 -2839.185,E2 -2839.185} C_VEL
LIN {X 0,Y 559.124,Z 614.953,A -85,B 0,C 180,E1 -2841.981,E2 -2841.981} C_VEL
LIN {X 0,Y 559.127,Z 614.958,A -85,B 0,C 180,E1 -2844.788,E2 -2844.788} C_VEL
LIN {X 0,Y 559.156,Z 614.961,A -85,B 0,C 180,E1 -2847.365,E2 -2847.365} C_VEL
LIN {X 0,Y 559.121,Z 614.956,A -85,B 0,C 180,E1 -2850.148,E2 -2850.148} C_VEL
LIN {X 0,Y 559.127,Z 614.957,A -85,B 0,C 180,E1 -2852.285,E2 -2852.285} C_VEL
LIN {X 0,Y 559.141,Z 614.956,A -85,B 0,C 180,E1 -2854.822,E2 -2854.822} C_VEL
LIN {X 0,Y 559.142,Z 614.958,A -85,B 0,C 180,E1 -2857.847,E2 -2857.847} C_VEL
LIN {X 0,Y 559.196,Z 614.947,A -85,B 0,C 180,E1 -2860.494,E2 -2860.494} C_VEL
LIN {X 0,Y 559.18,Z 614.952,A -85,B 0,C 180,E1 -2863.197,E2 -2863.197} C_VEL
LIN {X 0,Y 559.17,Z 614.953,A -85,B 0,C 180,E1 -2866.184,E2 -2866.184} C_VEL
LIN {X 0,Y 559.196,Z 614.949,A -85,B 0,C 180,E1 -2869.133,E2 -2869.133} C_VEL
LIN {X 0,Y 559.201,Z 614.951,A -85,B 0,C 180,E1 -2872.053,E2 -2872.053} C_VEL
LIN {X 0,Y 559.245,Z 614.942,A -85,B 0,C 180,E1 -2874.953,E2 -2874.953} C_VEL
LIN {X 0,Y 559.255,Z 614.95,A -85,B 0,C 180,E1 -2877.839,E2 -2877.839} C_VEL
LIN {X 0,Y 559.273,Z 614.937,A -85,B 0,C 180,E1 -2880.72,E2 -2880.72} C_VEL
LIN {X 0,Y 559.239,Z 614.943,A -85,B 0,C 180,E1 -2882.881,E2 -2882.881} C_VEL
LIN {X 0,Y 559.225,Z 614.952,A -85,B 0,C 180,E1 -2885.77,E2 -2885.77} C_VEL
LIN {X 0,Y 559.189,Z 614.95,A -85,B 0,C 180,E1 -2888.674,E2 -2888.674} C_VEL
LIN {X 0,Y 559.208,Z 614.949,A -85,B 0,C 180,E1 -2891.6,E2 -2891.6} C_VEL
LIN {X 0,Y 559.204,Z 614.948,A -85,B 0,C 180,E1 -2894.595,E2 -2894.595} C_VEL
LIN {X 0,Y 559.162,Z 614.954,A -85,B 0,C 180,E1 -2897.557,E2 -2897.557} C_VEL
LIN {X 0,Y 559.176,Z 614.955,A -85,B 0,C 180,E1 -2899.837,E2 -2899.837} C_VEL
LIN {X 0,Y 559.144,Z 614.965,A -85,B 0,C 180,E1 -2902.153,E2 -2902.153} C_VEL
LIN {X 0,Y 559.179,Z 614.95,A -85,B 0,C 180,E1 -2905.298,E2 -2905.298} C_VEL
LIN {X 0,Y 559.16,Z 614.954,A -85,B 0,C 180,E1 -2907.713,E2 -2907.713} C_VEL
LIN {X 0,Y 559.157,Z 614.961,A -85,B 0,C 180,E1 -2910.182,E2 -2910.182} C_VEL
LIN {X 0,Y 559.178,Z 614.954,A -85,B 0,C 180,E1 -2912.714,E2 -2912.714} C_VEL
LIN {X 0,Y 559.133,Z 614.956,A -85,B 0,C 180,E1 -2915.324,E2 -2915.324} C_VEL
LIN {X 0,Y 559.137,Z 614.959,A -85,B 0,C 180,E1 -2918.017,E2 -2918.017} C_VEL
LIN {X 0,Y 559.177,Z 614.955,A -85,B 0,C 180,E1 -2920.811,E2 -2920.811} C_VEL
LIN {X 0,Y 559.144,Z 614.955,A -85,B 0,C 180,E1 -2923.734,E2 -2923.734} C_VEL
LIN {X 0,Y 559.167,Z 614.958,A -85,B 0,C 180,E1 -2926.801,E2 -2926.801} C_VEL
LIN {X 0,Y 559.18,Z 614.952,A -85,B 0,C 180,E1 -2929.189,E2 -2929.189} C_VEL
LIN {X 0,Y 559.136,Z 614.957,A -85,B 0,C 180,E1 -2931.982,E2 -2931.982} C_VEL
LIN {X 0,Y 559.163,Z 614.962,A -85,B 0,C 180,E1 -2934.783,E2 -2934.783} C_VEL
LIN {X 0,Y 559.177,Z 614.953,A -85,B 0,C 180,E1 -2937.361,E2 -2937.361} C_VEL
LIN {X 0,Y 559.152,Z 614.956,A -85,B 0,C 180,E1 -2940.142,E2 -2940.142} C_VEL
LIN {X 0,Y 559.185,Z 614.958,A -85,B 0,C 180,E1 -2943.17,E2 -2943.17} C_VEL
LIN {X 0,Y 559.221,Z 615.119,A -85,B 0,C 180,E1 -2944.579,E2 -2944.579} C_VEL
LIN {X 0,Y 560.643,Z 621.803,A -85,B 0,C 180,E1 -2945.564,E2 -2945.564} C_VEL
LIN {X 0,Y 560.374,Z 639.14,A -85,B 0,C 180,E1 -2947.898,E2 -2947.898} C_VEL
LIN {X 0,Y 559.983,Z 659.702,A -85,B 0,C 180,E1 -2950.618,E2 -2950.618} C_VEL
LIN {X 0,Y 559.762,Z 676.392,A -85,B 0,C 180,E1 -2952.799,E2 -2952.799} C_VEL
LIN {X 0,Y 561.019,Z 684.077,A -85,B 0,C 180,E1 -2952.948,E2 -2952.948} C_VEL
LIN {X 0,Y 560.581,Z 814.879,A -85,B 0,C 180,E1 -2954.665,E2 -2954.665} C_VEL
LIN {X 0,Y 560.405,Z 829.139,A -85,B 0,C 180,E1 -2955.002,E2 -2955.002} C_VEL
LIN {X 0,Y 560.247,Z 842.707,A -85,B 0,C 180,E1 -2955.47,E2 -2955.47} C_VEL
LIN {X 0,Y 560.055,Z 856.641,A -85,B 0,C 180,E1 -2956.114,E2 -2956.114} C_VEL
LIN {X 0,Y 559.841,Z 869.099,A -85,B 0,C 180,E1 -2956.848,E2 -2956.848} C_VEL
LIN {X 0,Y 559.617,Z 880.479,A -85,B 0,C 180,E1 -2957.673,E2 -2957.673} C_VEL
LIN {X 0,Y 559.454,Z 891.643,A -85,B 0,C 180,E1 -2958.655,E2 -2958.655} C_VEL
LIN {X 0,Y 559.239,Z 901.332,A -85,B 0,C 180,E1 -2959.684,E2 -2959.684} C_VEL
LIN {X 0,Y 559.114,Z 909.911,A -85,B 0,C 180,E1 -2960.778,E2 -2960.778} C_VEL
LIN {X 0,Y 558.979,Z 918.115,A -85,B 0,C 180,E1 -2962.05,E2 -2962.05} C_VEL
LIN {X 0,Y 558.894,Z 925.165,A -85,B 0,C 180,E1 -2963.42,E2 -2963.42} C_VEL
LIN {X 0,Y 558.858,Z 929.961,A -85,B 0,C 180,E1 -2964.588,E2 -2964.588} C_VEL
LIN {X 0,Y 558.866,Z 933.443,A -85,B 0,C 180,E1 -2965.673,E2 -2965.673} C_VEL
LIN {X 0,Y 558.796,Z 936.832,A -85,B 0,C 180,E1 -2967.116,E2 -2967.116} C_VEL
LIN {X 0,Y 558.74,Z 938.833,A -85,B 0,C 180,E1 -2968.558,E2 -2968.558} C_VEL
LIN {X 0,Y 558.738,Z 939.5,A -85,B 0,C 180,E1 -2970,E2 -2970} C_VEL
LIN {X 0,Y 558.74,Z 938.834,A -85,B 0,C 180,E1 -2971.441,E2 -2971.441} C_VEL
LIN {X 0,Y 558.795,Z 936.834,A -85,B 0,C 180,E1 -2972.884,E2 -2972.884} C_VEL
LIN {X 0,Y 558.866,Z 933.445,A -85,B 0,C 180,E1 -2974.327,E2 -2974.327} C_VEL
LIN {X 0,Y 558.917,Z 928.568,A -85,B 0,C 180,E1 -2975.773,E2 -2975.773} C_VEL
LIN {X 0,Y 558.907,Z 922.053,A -85,B 0,C 180,E1 -2977.224,E2 -2977.224} C_VEL
LIN {X 0,Y 559.028,Z 914.801,A -85,B 0,C 180,E1 -2978.495,E2 -2978.495} C_VEL
LIN {X 0,Y 559.146,Z 905.823,A -85,B 0,C 180,E1 -2979.769,E2 -2979.769} C_VEL
LIN {X 0,Y 559.35,Z 896.392,A -85,B 0,C 180,E1 -2980.863,E2 -2980.863} C_VEL
LIN {X 0,Y 559.521,Z 885.951,A -85,B 0,C 180,E1 -2981.869,E2 -2981.869} C_VEL
LIN {X 0,Y 559.715,Z 874.435,A -85,B 0,C 180,E1 -2982.786,E2 -2982.786} C_VEL
LIN {X 0,Y 559.951,Z 861.645,A -85,B 0,C 180,E1 -2983.611,E2 -2983.611} C_VEL
LIN {X 0,Y 560.185,Z 849.154,A -85,B 0,C 180,E1 -2984.253,E2 -2984.253} C_VEL
LIN {X 0,Y 560.372,Z 835.275,A -85,B 0,C 180,E1 -2984.804,E2 -2984.804} C_VEL
LIN {X 0,Y 560.511,Z 821.631,A -85,B 0,C 180,E1 -2985.194,E2 -2985.194} C_VEL
LIN {X 0,Y 560.608,Z 807.603,A -85,B 0,C 180,E1 -2985.45,E2 -2985.45} C_VEL
LIN {X 0,Y 561.004,Z 684.089,A -85,B 0,C 180,E1 -2987.052,E2 -2987.052} C_VEL
LIN {X 0,Y 559.736,Z 676.455,A -85,B 0,C 180,E1 -2987.194,E2 -2987.194} C_VEL
LIN {X 0,Y 560.074,Z 655.032,A -85,B 0,C 180,E1 -2989.995,E2 -2989.995} C_VEL
LIN {X 0,Y 560.521,Z 631.917,A -85,B 0,C 180,E1 -2993.068,E2 -2993.068} C_VEL
LIN {X 0,Y 560.642,Z 621.804,A -85,B 0,C 180,E1 -2994.436,E2 -2994.436} C_VEL
LIN {X 0,Y 559.175,Z 614.959,A -85,B 0,C 180,E1 -2995.448,E2 -2995.448} C_VEL
LIN {X 0,Y 559.172,Z 614.954,A -85,B 0,C 180,E1 -2998.382,E2 -2998.382} C_VEL
LIN {X 0,Y 559.155,Z 614.962,A -85,B 0,C 180,E1 -3001.275,E2 -3001.275} C_VEL
LIN {X 0,Y 559.17,Z 614.952,A -85,B 0,C 180,E1 -3003.95,E2 -3003.95} C_VEL
LIN {X 0,Y 559.171,Z 614.951,A -85,B 0,C 180,E1 -3006.449,E2 -3006.449} C_VEL
LIN {X 0,Y 559.18,Z 614.953,A -85,B 0,C 180,E1 -3008.934,E2 -3008.934} C_VEL
LIN {X 0,Y 559.194,Z 614.954,A -85,B 0,C 180,E1 -3011.767,E2 -3011.767} C_VEL
LIN {X 0,Y 559.141,Z 614.955,A -85,B 0,C 180,E1 -3014.739,E2 -3014.739} C_VEL
LIN {X 0,Y 559.178,Z 614.954,A -85,B 0,C 180,E1 -3017.863,E2 -3017.863} C_VEL
LIN {X 0,Y 559.187,Z 614.952,A -85,B 0,C 180,E1 -3020.135,E2 -3020.135} C_VEL
LIN {X 0,Y 559.148,Z 614.951,A -85,B 0,C 180,E1 -3022.892,E2 -3022.892} C_VEL
LIN {X 0,Y 559.16,Z 614.961,A -85,B 0,C 180,E1 -3025.556,E2 -3025.556} C_VEL
LIN {X 0,Y 559.173,Z 614.95,A -85,B 0,C 180,E1 -3028.138,E2 -3028.138} C_VEL
LIN {X 0,Y 559.145,Z 614.954,A -85,B 0,C 180,E1 -3030.646,E2 -3030.646} C_VEL
LIN {X 0,Y 559.173,Z 614.952,A -85,B 0,C 180,E1 -3033.172,E2 -3033.172} C_VEL
LIN {X 0,Y 559.159,Z 614.956,A -85,B 0,C 180,E1 -3035.495,E2 -3035.495} C_VEL
LIN {X 0,Y 559.174,Z 614.952,A -85,B 0,C 180,E1 -3038.624,E2 -3038.624} C_VEL
LIN {X 0,Y 559.173,Z 614.95,A -85,B 0,C 180,E1 -3040.927,E2 -3040.927} C_VEL
LIN {X 0,Y 559.172,Z 614.96,A -85,B 0,C 180,E1 -3043.948,E2 -3043.948} C_VEL
LIN {X 0,Y 559.174,Z 614.959,A -85,B 0,C 180,E1 -3046.184,E2 -3046.184} C_VEL
LIN {X 0,Y 559.199,Z 614.948,A -85,B 0,C 180,E1 -3049.134,E2 -3049.134} C_VEL
LIN {X 0,Y 559.202,Z 614.954,A -85,B 0,C 180,E1 -3052.054,E2 -3052.054} C_VEL
LIN {X 0,Y 559.255,Z 614.94,A -85,B 0,C 180,E1 -3054.954,E2 -3054.954} C_VEL
LIN {X 0,Y 559.253,Z 614.944,A -85,B 0,C 180,E1 -3057.84,E2 -3057.84} C_VEL
LIN {X 0,Y 559.271,Z 614.942,A -85,B 0,C 180,E1 -3060.72,E2 -3060.72} C_VEL
LIN {X 0,Y 559.237,Z 614.946,A -85,B 0,C 180,E1 -3062.882,E2 -3062.882} C_VEL
LIN {X 0,Y 559.232,Z 614.943,A -85,B 0,C 180,E1 -3065.77,E2 -3065.77} C_VEL
LIN {X 0,Y 559.187,Z 614.956,A -85,B 0,C 180,E1 -3068.675,E2 -3068.675} C_VEL
LIN {X 0,Y 559.208,Z 614.946,A -85,B 0,C 180,E1 -3071.601,E2 -3071.601} C_VEL
LIN {X 0,Y 559.203,Z 614.956,A -85,B 0,C 180,E1 -3074.596,E2 -3074.596} C_VEL
LIN {X 0,Y 559.145,Z 614.955,A -85,B 0,C 180,E1 -3077.558,E2 -3077.558} C_VEL
LIN {X 0,Y 559.168,Z 614.95,A -85,B 0,C 180,E1 -3079.838,E2 -3079.838} C_VEL
LIN {X 0,Y 559.142,Z 614.957,A -85,B 0,C 180,E1 -3082.153,E2 -3082.153} C_VEL
LIN {X 0,Y 559.177,Z 614.953,A -85,B 0,C 180,E1 -3085.298,E2 -3085.298} C_VEL
LIN {X 0,Y 559.13,Z 614.954,A -85,B 0,C 180,E1 -3087.715,E2 -3087.715} C_VEL
LIN {X 0,Y 559.137,Z 614.957,A -85,B 0,C 180,E1 -3090.616,E2 -3090.616} C_VEL
LIN {X 0,Y 558.476,Z 615.047,A -85,B 0,C 180,E1 -3091.218,E2 -3091.218} C_VEL
LIN {X 0,Y 555.613,Z 615.403,A -85,B 0,C 180,E1 -3092.194,E2 -3092.194} C_VEL
LIN {X 0,Y 553.196,Z 615.705,A -85,B 0,C 180,E1 -3092.98,E2 -3092.98} C_VEL
LIN {X 0,Y 552.168,Z 615.825,A -85,B 0,C 180,E1 -3093.586,E2 -3093.586} C_VEL
LIN {X 0,Y 552.091,Z 615.833,A -85,B 0,C 180,E1 -3093.792,E2 -3093.792} C_VEL
LIN {X 0,Y 552.108,Z 615.837,A -85,B 0,C 180,E1 -3096.747,E2 -3096.747} C_VEL
LIN {X 0,Y 552.13,Z 615.83,A -85,B 0,C 180,E1 -3099.528,E2 -3099.528} C_VEL
LIN {X 0,Y 552.11,Z 615.832,A -85,B 0,C 180,E1 -3102.428,E2 -3102.428} C_VEL
LIN {X 0,Y 552.077,Z 615.839,A -85,B 0,C 180,E1 -3105.56,E2 -3105.56} C_VEL
LIN {X 0,Y 552.079,Z 615.838,A -85,B 0,C 180,E1 -3108.684,E2 -3108.684} C_VEL
LIN {X 0,Y 552.116,Z 615.84,A -85,B 0,C 180,E1 -3111.411,E2 -3111.411} C_VEL
LIN {X 0,Y 552.078,Z 615.835,A -85,B 0,C 180,E1 -3114.156,E2 -3114.156} C_VEL
LIN {X 0,Y 552.11,Z 615.836,A -85,B 0,C 180,E1 -3117.155,E2 -3117.155} C_VEL
LIN {X 0,Y 552.097,Z 615.837,A -85,B 0,C 180,E1 -3119.954,E2 -3119.954} C_VEL
LIN {X 0,Y 552.079,Z 615.841,A -85,B 0,C 180,E1 -3123.013,E2 -3123.013} C_VEL
LIN {X 0,Y 552.145,Z 615.897,A -85,B 0,C 180,E1 -3123.824,E2 -3123.824} C_VEL
LIN {X 0,Y 552.827,Z 621.707,A -85,B 0,C 180,E1 -3124.818,E2 -3124.818} C_VEL
LIN {X 0,Y 552.536,Z 638.913,A -85,B 0,C 180,E1 -3127.637,E2 -3127.637} C_VEL
LIN {X 0,Y 554.21,Z 648.146,A -85,B 0,C 180,E1 -3127.818,E2 -3127.818} C_VEL
LIN {X 0,Y 553.774,Z 775.04,A -85,B 0,C 180,E1 -3129.501,E2 -3129.501} C_VEL
LIN {X 0,Y 553.59,Z 789.318,A -85,B 0,C 180,E1 -3129.833,E2 -3129.833} C_VEL
LIN {X 0,Y 553.381,Z 803.795,A -85,B 0,C 180,E1 -3130.334,E2 -3130.334} C_VEL
LIN {X 0,Y 553.174,Z 816.167,A -85,B 0,C 180,E1 -3130.904,E2 -3130.904} C_VEL
LIN {X 0,Y 552.916,Z 827.707,A -85,B 0,C 180,E1 -3131.568,E2 -3131.568} C_VEL
LIN {X 0,Y 552.705,Z 839.075,A -85,B 0,C 180,E1 -3132.369,E2 -3132.369} C_VEL
LIN {X 0,Y 552.448,Z 850.688,A -85,B 0,C 180,E1 -3133.367,E2 -3133.367} C_VEL
LIN {X 0,Y 552.229,Z 861.478,A -85,B 0,C 180,E1 -3134.499,E2 -3134.499} C_VEL
LIN {X 0,Y 552.029,Z 870.731,A -85,B 0,C 180,E1 -3135.679,E2 -3135.679} C_VEL
LIN {X 0,Y 551.888,Z 878.802,A -85,B 0,C 180,E1 -3136.936,E2 -3136.936} C_VEL
LIN {X 0,Y 551.804,Z 885.555,A -85,B 0,C 180,E1 -3138.242,E2 -3138.242} C_VEL
LIN {X 0,Y 551.745,Z 891.518,A -85,B 0,C 180,E1 -3139.728,E2 -3139.728} C_VEL
LIN {X 0,Y 551.694,Z 895.867,A -85,B 0,C 180,E1 -3141.207,E2 -3141.207} C_VEL
LIN {X 0,Y 551.694,Z 898.741,A -85,B 0,C 180,E1 -3142.681,E2 -3142.681} C_VEL
LIN {X 0,Y 551.707,Z 900.23,A -85,B 0,C 180,E1 -3144.151,E2 -3144.151} C_VEL
LIN {X 0,Y 551.695,Z 900.383,A -85,B 0,C 180,E1 -3145.616,E2 -3145.616} C_VEL
LIN {X 0,Y 551.712,Z 899.21,A -85,B 0,C 180,E1 -3147.079,E2 -3147.079} C_VEL
LIN {X 0,Y 551.649,Z 896.691,A -85,B 0,C 180,E1 -3148.54,E2 -3148.54} C_VEL
LIN {X 0,Y 551.686,Z 892.744,A -85,B 0,C 180,E1 -3150,E2 -3150} C_VEL
LIN {X 0,Y 551.825,Z 888.786,A -85,B 0,C 180,E1 -3151.095,E2 -3151.095} C_VEL
LIN {X 0,Y 551.77,Z 883.905,A -85,B 0,C 180,E1 -3152.19,E2 -3152.19} C_VEL
LIN {X 0,Y 551.951,Z 876.905,A -85,B 0,C 180,E1 -3153.468,E2 -3153.468} C_VEL
LIN {X 0,Y 552.13,Z 868.266,A -85,B 0,C 180,E1 -3154.746,E2 -3154.746} C_VEL
LIN {X 0,Y 552.305,Z 859.257,A -85,B 0,C 180,E1 -3155.843,E2 -3155.843} C_VEL
LIN {X 0,Y 552.506,Z 849.025,A -85,B 0,C 180,E1 -3156.88,E2 -3156.88} C_VEL
LIN {X 0,Y 552.753,Z 837.331,A -85,B 0,C 180,E1 -3157.856,E2 -3157.856} C_VEL
LIN {X 0,Y 553.013,Z 825.168,A -85,B 0,C 180,E1 -3158.68,E2 -3158.68} C_VEL
LIN {X 0,Y 553.192,Z 813.536,A -85,B 0,C 180,E1 -3159.322,E2 -3159.322} C_VEL
LIN {X 0,Y 553.451,Z 799.641,A -85,B 0,C 180,E1 -3159.917,E2 -3159.917} C_VEL
LIN {X 0,Y 553.615,Z 785.753,A -85,B 0,C 180,E1 -3160.353,E2 -3160.353} C_VEL
LIN {X 0,Y 553.76,Z 771.187,A -85,B 0,C 180,E1 -3160.651,E2 -3160.651} C_VEL
LIN {X 0,Y 554.103,Z 646.945,A -85,B 0,C 180,E1 -3162.292,E2 -3162.292} C_VEL
LIN {X 0,Y 552.553,Z 638.864,A -85,B 0,C 180,E1 -3162.461,E2 -3162.461} C_VEL
LIN {X 0,Y 552.863,Z 621.489,A -85,B 0,C 180,E1 -3165.307,E2 -3165.307} C_VEL
LIN {X 0,Y 552.113,Z 615.84,A -85,B 0,C 180,E1 -3166.31,E2 -3166.31} C_VEL
LIN {X 0,Y 552.119,Z 615.832,A -85,B 0,C 180,E1 -3169.616,E2 -3169.616} C_VEL
LIN {X 0,Y 552.086,Z 615.842,A -85,B 0,C 180,E1 -3172.451,E2 -3172.451} C_VEL
LIN {X 0,Y 552.064,Z 615.839,A -85,B 0,C 180,E1 -3175.329,E2 -3175.329} C_VEL
LIN {X 0,Y 552.055,Z 615.84,A -85,B 0,C 180,E1 -3178.102,E2 -3178.102} C_VEL
LIN {X 0,Y 552.077,Z 615.843,A -85,B 0,C 180,E1 -3180.611,E2 -3180.611} C_VEL
LIN {X 0,Y 552.092,Z 615.838,A -85,B 0,C 180,E1 -3183.188,E2 -3183.188} C_VEL
LIN {X 0,Y 552.071,Z 615.836,A -85,B 0,C 180,E1 -3185.845,E2 -3185.845} C_VEL
LIN {X 0,Y 552.113,Z 615.835,A -85,B 0,C 180,E1 -3188.59,E2 -3188.59} C_VEL
LIN {X 0,Y 552.066,Z 615.839,A -85,B 0,C 180,E1 -3191.451,E2 -3191.451} C_VEL
LIN {X 0,Y 552.078,Z 615.837,A -85,B 0,C 180,E1 -3194.529,E2 -3194.529} C_VEL
LIN {X 0,Y 552.085,Z 615.836,A -85,B 0,C 180,E1 -3197.59,E2 -3197.59} C_VEL
LIN {X 0,Y 552.111,Z 615.831,A -85,B 0,C 180,E1 -3200.471,E2 -3200.471} C_VEL
LIN {X 0,Y 552.099,Z 615.837,A -85,B 0,C 180,E1 -3203.318,E2 -3203.318} C_VEL
LIN {X 0,Y 552.102,Z 615.833,A -85,B 0,C 180,E1 -3205.937,E2 -3205.937} C_VEL
LIN {X 0,Y 552.124,Z 615.829,A -85,B 0,C 180,E1 -3208.54,E2 -3208.54} C_VEL
LIN {X 0,Y 552.098,Z 615.84,A -85,B 0,C 180,E1 -3211.444,E2 -3211.444} C_VEL
LIN {X 0,Y 552.08,Z 615.834,A -85,B 0,C 180,E1 -3214.353,E2 -3214.353} C_VEL
LIN {X 0,Y 552.096,Z 615.831,A -85,B 0,C 180,E1 -3216.757,E2 -3216.757} C_VEL
LIN {X 0,Y 552.121,Z 615.834,A -85,B 0,C 180,E1 -3219.12,E2 -3219.12} C_VEL
LIN {X 0,Y 552.119,Z 615.838,A -85,B 0,C 180,E1 -3221.444,E2 -3221.444} C_VEL
LIN {X 0,Y 552.113,Z 615.836,A -85,B 0,C 180,E1 -3223.737,E2 -3223.737} C_VEL
LIN {X 0,Y 552.135,Z 615.831,A -85,B 0,C 180,E1 -3226.004,E2 -3226.004} C_VEL
LIN {X 0,Y 552.165,Z 615.823,A -85,B 0,C 180,E1 -3228.993,E2 -3228.993} C_VEL
LIN {X 0,Y 552.156,Z 615.83,A -85,B 0,C 180,E1 -3231.951,E2 -3231.951} C_VEL
LIN {X 0,Y 552.22,Z 615.817,A -85,B 0,C 180,E1 -3234.889,E2 -3234.889} C_VEL
LIN {X 0,Y 552.226,Z 615.826,A -85,B 0,C 180,E1 -3237.812,E2 -3237.812} C_VEL
LIN {X 0,Y 552.243,Z 615.813,A -85,B 0,C 180,E1 -3240.729,E2 -3240.729} C_VEL
LIN {X 0,Y 552.206,Z 615.819,A -85,B 0,C 180,E1 -3242.918,E2 -3242.918} C_VEL
LIN {X 0,Y 552.195,Z 615.829,A -85,B 0,C 180,E1 -3245.844,E2 -3245.844} C_VEL
LIN {X 0,Y 552.156,Z 615.825,A -85,B 0,C 180,E1 -3248.786,E2 -3248.786} C_VEL
LIN {X 0,Y 552.166,Z 615.829,A -85,B 0,C 180,E1 -3251.75,E2 -3251.75} C_VEL
LIN {X 0,Y 552.14,Z 615.827,A -85,B 0,C 180,E1 -3254.748,E2 -3254.748} C_VEL
LIN {X 0,Y 552.113,Z 615.835,A -85,B 0,C 180,E1 -3257.788,E2 -3257.788} C_VEL
LIN {X 0,Y 552.134,Z 615.836,A -85,B 0,C 180,E1 -3260.101,E2 -3260.101} C_VEL
LIN {X 0,Y 552.095,Z 615.837,A -85,B 0,C 180,E1 -3262.451,E2 -3262.451} C_VEL
LIN {X 0,Y 552.158,Z 615.825,A -85,B 0,C 180,E1 -3265.35,E2 -3265.35} C_VEL
LIN {X 0,Y 552.112,Z 615.837,A -85,B 0,C 180,E1 -3268.098,E2 -3268.098} C_VEL
LIN {X 0,Y 552.107,Z 615.836,A -85,B 0,C 180,E1 -3270.609,E2 -3270.609} C_VEL
LIN {X 0,Y 552.126,Z 615.829,A -85,B 0,C 180,E1 -3273.185,E2 -3273.185} C_VEL
LIN {X 0,Y 552.089,Z 615.836,A -85,B 0,C 180,E1 -3275.843,E2 -3275.843} C_VEL
LIN {X 0,Y 552.128,Z 615.83,A -85,B 0,C 180,E1 -3279.062,E2 -3279.062} C_VEL
LIN {X 0,Y 552.133,Z 615.828,A -85,B 0,C 180,E1 -3281.445,E2 -3281.445} C_VEL
LIN {X 0,Y 552.098,Z 615.842,A -85,B 0,C 180,E1 -3284.532,E2 -3284.532} C_VEL
LIN {X 0,Y 552.133,Z 615.828,A -85,B 0,C 180,E1 -3287.584,E2 -3287.584} C_VEL
LIN {X 0,Y 552.131,Z 615.836,A -85,B 0,C 180,E1 -3290.473,E2 -3290.473} C_VEL
LIN {X 0,Y 552.117,Z 615.832,A -85,B 0,C 180,E1 -3293.316,E2 -3293.316} C_VEL
LIN {X 0,Y 552.134,Z 615.829,A -85,B 0,C 180,E1 -3295.939,E2 -3295.939} C_VEL
LIN {X 0,Y 552.121,Z 615.837,A -85,B 0,C 180,E1 -3298.541,E2 -3298.541} C_VEL
LIN {X 0,Y 552.127,Z 615.833,A -85,B 0,C 180,E1 -3301.438,E2 -3301.438} C_VEL
LIN {X 0,Y 552.193,Z 615.986,A -85,B 0,C 180,E1 -3304.385,E2 -3304.385} C_VEL
LIN {X 0,Y 553.764,Z 623.351,A -85,B 0,C 180,E1 -3305.46,E2 -3305.46} C_VEL
LIN {X 0,Y 553.505,Z 640.468,A -85,B 0,C 180,E1 -3307.79,E2 -3307.79} C_VEL
LIN {X 0,Y 553.038,Z 663.699,A -85,B 0,C 180,E1 -3310.899,E2 -3310.899} C_VEL
LIN {X 0,Y 552.792,Z 676.402,A -85,B 0,C 180,E1 -3312.577,E2 -3312.577} C_VEL
LIN {X 0,Y 554.255,Z 685.853,A -85,B 0,C 180,E1 -3312.757,E2 -3312.757} C_VEL
LIN {X 0,Y 553.746,Z 814.878,A -85,B 0,C 180,E1 -3314.471,E2 -3314.471} C_VEL
LIN {X 0,Y 553.54,Z 829.237,A -85,B 0,C 180,E1 -3314.815,E2 -3314.815} C_VEL
LIN {X 0,Y 553.369,Z 842.706,A -85,B 0,C 180,E1 -3315.285,E2 -3315.285} C_VEL
LIN {X 0,Y 553.156,Z 856.64,A -85,B 0,C 180,E1 -3315.937,E2 -3315.937} C_VEL
LIN {X 0,Y 552.896,Z 869.101,A -85,B 0,C 180,E1 -3316.68,E2 -3316.68} C_VEL
LIN {X 0,Y 552.655,Z 880.481,A -85,B 0,C 180,E1 -3317.515,E2 -3317.515} C_VEL
LIN {X 0,Y 552.413,Z 890.649,A -85,B 0,C 180,E1 -3318.413,E2 -3318.413} C_VEL
LIN {X 0,Y 552.227,Z 901.332,A -85,B 0,C 180,E1 -3319.551,E2 -3319.551} C_VEL
LIN {X 0,Y 552.071,Z 909.911,A -85,B 0,C 180,E1 -3320.659,E2 -3320.659} C_VEL
LIN {X 0,Y 551.901,Z 918.116,A -85,B 0,C 180,E1 -3321.948,E2 -3321.948} C_VEL
LIN {X 0,Y 551.823,Z 923.863,A -85,B 0,C 180,E1 -3323.051,E2 -3323.051} C_VEL
LIN {X 0,Y 551.791,Z 929.961,A -85,B 0,C 180,E1 -3324.518,E2 -3324.518} C_VEL
LIN {X 0,Y 551.76,Z 933.443,A -85,B 0,C 180,E1 -3325.617,E2 -3325.617} C_VEL
LIN {X 0,Y 551.72,Z 936.832,A -85,B 0,C 180,E1 -3327.079,E2 -3327.079} C_VEL
LIN {X 0,Y 551.64,Z 938.833,A -85,B 0,C 180,E1 -3328.54,E2 -3328.54} C_VEL
LIN {X 0,Y 551.639,Z 939.5,A -85,B 0,C 180,E1 -3330,E2 -3330} C_VEL
LIN {X 0,Y 551.64,Z 938.834,A -85,B 0,C 180,E1 -3331.46,E2 -3331.46} C_VEL
LIN {X 0,Y 551.72,Z 936.834,A -85,B 0,C 180,E1 -3332.921,E2 -3332.921} C_VEL
LIN {X 0,Y 551.76,Z 933.446,A -85,B 0,C 180,E1 -3334.383,E2 -3334.383} C_VEL
LIN {X 0,Y 551.825,Z 928.568,A -85,B 0,C 180,E1 -3335.848,E2 -3335.848} C_VEL
LIN {X 0,Y 551.832,Z 922.054,A -85,B 0,C 180,E1 -3337.317,E2 -3337.317} C_VEL
LIN {X 0,Y 551.962,Z 914.802,A -85,B 0,C 180,E1 -3338.604,E2 -3338.604} C_VEL
LIN {X 0,Y 552.116,Z 905.823,A -85,B 0,C 180,E1 -3339.895,E2 -3339.895} C_VEL
LIN {X 0,Y 552.346,Z 896.392,A -85,B 0,C 180,E1 -3341.003,E2 -3341.003} C_VEL
LIN {X 0,Y 552.543,Z 885.952,A -85,B 0,C 180,E1 -3342.022,E2 -3342.022} C_VEL
LIN {X 0,Y 552.776,Z 874.435,A -85,B 0,C 180,E1 -3342.949,E2 -3342.949} C_VEL
LIN {X 0,Y 553.04,Z 861.643,A -85,B 0,C 180,E1 -3343.785,E2 -3343.785} C_VEL
LIN {X 0,Y 553.302,Z 849.152,A -85,B 0,C 180,E1 -3344.435,E2 -3344.435} C_VEL
LIN {X 0,Y 553.501,Z 836.026,A -85,B 0,C 180,E1 -3344.965,E2 -3344.965} C_VEL
LIN {X 0,Y 553.653,Z 821.907,A -85,B 0,C 180,E1 -3345.38,E2 -3345.38} C_VEL
LIN {X 0,Y 553.774,Z 807.603,A -85,B 0,C 180,E1 -3345.646,E2 -3345.646} C_VEL
LIN {X 0,Y 554.129,Z 683.744,A -85,B 0,C 180,E1 -3347.275,E2 -3347.275} C_VEL
LIN {X 0,Y 552.807,Z 676.295,A -85,B 0,C 180,E1 -3347.437,E2 -3347.437} C_VEL
LIN {X 0,Y 553.221,Z 653.588,A -85,B 0,C 180,E1 -3350.448,E2 -3350.448} C_VEL
LIN {X 0,Y 553.667,Z 631.938,A -85,B 0,C 180,E1 -3353.367,E2 -3353.367} C_VEL
LIN {X 0,Y 553.737,Z 623.203,A -85,B 0,C 180,E1 -3354.561,E2 -3354.561} C_VEL
LIN {X 0,Y 552.181,Z 615.83,A -85,B 0,C 180,E1 -3355.642,E2 -3355.642} C_VEL
LIN {X 0,Y 552.128,Z 615.833,A -85,B 0,C 180,E1 -3358.562,E2 -3358.562} C_VEL
LIN {X 0,Y 552.137,Z 615.834,A -85,B 0,C 180,E1 -3361.48,E2 -3361.48} C_VEL
LIN {X 0,Y 552.14,Z 615.827,A -85,B 0,C 180,E1 -3364.171,E2 -3364.171} C_VEL
LIN {X 0,Y 552.114,Z 615.832,A -85,B 0,C 180,E1 -3366.746,E2 -3366.746} C_VEL
LIN {X 0,Y 552.136,Z 615.835,A -85,B 0,C 180,E1 -3369.527,E2 -3369.527} C_VEL
LIN {X 0,Y 552.132,Z 615.828,A -85,B 0,C 180,E1 -3372.425,E2 -3372.425} C_VEL
LIN {X 0,Y 552.1,Z 615.842,A -85,B 0,C 180,E1 -3375.563,E2 -3375.563} C_VEL
LIN {X 0,Y 552.142,Z 615.825,A -85,B 0,C 180,E1 -3378.676,E2 -3378.676} C_VEL
LIN {X 0,Y 552.122,Z 615.836,A -85,B 0,C 180,E1 -3381.411,E2 -3381.411} C_VEL
LIN {X 0,Y 552.115,Z 615.833,A -85,B 0,C 180,E1 -3384.159,E2 -3384.159} C_VEL
LIN {X 0,Y 552.125,Z 615.828,A -85,B 0,C 180,E1 -3386.815,E2 -3386.815} C_VEL
LIN {X 0,Y 552.109,Z 615.83,A -85,B 0,C 180,E1 -3389.391,E2 -3389.391} C_VEL
LIN {X 0,Y 552.128,Z 615.837,A -85,B 0,C 180,E1 -3391.903,E2 -3391.903} C_VEL
LIN {X 0,Y 552.157,Z 615.825,A -85,B 0,C 180,E1 -3394.65,E2 -3394.65} C_VEL
LIN {X 0,Y 552.098,Z 615.836,A -85,B 0,C 180,E1 -3397.549,E2 -3397.549} C_VEL
LIN {X 0,Y 552.159,Z 615.825,A -85,B 0,C 180,E1 -3400.675,E2 -3400.675} C_VEL
LIN {X 0,Y 552.122,Z 615.834,A -85,B 0,C 180,E1 -3403.738,E2 -3403.738} C_VEL
LIN {X 0,Y 552.138,Z 615.836,A -85,B 0,C 180,E1 -3406.005,E2 -3406.005} C_VEL
LIN {X 0,Y 552.166,Z 615.824,A -85,B 0,C 180,E1 -3408.994,E2 -3408.994} C_VEL
LIN {X 0,Y 552.157,Z 615.829,A -85,B 0,C 180,E1 -3411.952,E2 -3411.952} C_VEL
LIN {X 0,Y 552.23,Z 615.816,A -85,B 0,C 180,E1 -3414.889,E2 -3414.889} C_VEL
LIN {X 0,Y 552.225,Z 615.819,A -85,B 0,C 180,E1 -3417.812,E2 -3417.812} C_VEL
LIN {X 0,Y 552.242,Z 615.817,A -85,B 0,C 180,E1 -3420.729,E2 -3420.729} C_VEL
LIN {X 0,Y 552.204,Z 615.822,A -85,B 0,C 180,E1 -3422.918,E2 -3422.918} C_VEL
LIN {X 0,Y 552.202,Z 615.819,A -85,B 0,C 180,E1 -3425.844,E2 -3425.844} C_VEL
LIN {X 0,Y 552.155,Z 615.83,A -85,B 0,C 180,E1 -3428.786,E2 -3428.786} C_VEL
LIN {X 0,Y 552.165,Z 615.824,A -85,B 0,C 180,E1 -3431.751,E2 -3431.751} C_VEL
LIN {X 0,Y 552.139,Z 615.834,A -85,B 0,C 180,E1 -3434.749,E2 -3434.749} C_VEL
LIN {X 0,Y 552.102,Z 615.832,A -85,B 0,C 180,E1 -3437.789,E2 -3437.789} C_VEL
LIN {X 0,Y 552.129,Z 615.829,A -85,B 0,C 180,E1 -3440.102,E2 -3440.102} C_VEL
LIN {X 0,Y 552.093,Z 615.838,A -85,B 0,C 180,E1 -3442.451,E2 -3442.451} C_VEL
LIN {X 0,Y 552.139,Z 615.83,A -85,B 0,C 180,E1 -3445.346,E2 -3445.346} C_VEL
LIN {X 0,Y 552.08,Z 615.833,A -85,B 0,C 180,E1 -3448.1,E2 -3448.1} C_VEL
LIN {X 0,Y 552.101,Z 615.834,A -85,B 0,C 180,E1 -3450.613,E2 -3450.613} C_VEL
LIN {X 0,Y 552.108,Z 615.836,A -85,B 0,C 180,E1 -3453.187,E2 -3453.187} C_VEL
LIN {X 0,Y 552.091,Z 615.833,A -85,B 0,C 180,E1 -3453.792,E2 -3453.792} C_VEL
LIN {X 0,Y 551.451,Z 615.915,A -85,B 0,C 180,E1 -3454.4,E2 -3454.4} C_VEL
LIN {X 0,Y 548.637,Z 616.27,A -85,B 0,C 180,E1 -3455.389,E2 -3455.389} C_VEL
LIN {X 0,Y 546.228,Z 616.574,A -85,B 0,C 180,E1 -3456.184,E2 -3456.184} C_VEL
LIN {X 0,Y 545.165,Z 616.706,A -85,B 0,C 180,E1 -3456.798,E2 -3456.798} C_VEL
LIN {X 0,Y 545.063,Z 616.717,A -85,B 0,C 180,E1 -3457.006,E2 -3457.006} C_VEL
LIN {X 0,Y 545.066,Z 616.707,A -85,B 0,C 180,E1 -3460.143,E2 -3460.143} C_VEL
LIN {X 0,Y 545.025,Z 616.723,A -85,B 0,C 180,E1 -3463.112,E2 -3463.112} C_VEL
LIN {X 0,Y 545.048,Z 616.711,A -85,B 0,C 180,E1 -3466.227,E2 -3466.227} C_VEL
LIN {X 0,Y 545.03,Z 616.718,A -85,B 0,C 180,E1 -3468.881,E2 -3468.881} C_VEL
LIN {X 0,Y 545.05,Z 616.715,A -85,B 0,C 180,E1 -3471.762,E2 -3471.762} C_VEL
LIN {X 0,Y 545.03,Z 616.713,A -85,B 0,C 180,E1 -3474.531,E2 -3474.531} C_VEL
LIN {X 0,Y 545.065,Z 616.713,A -85,B 0,C 180,E1 -3477.211,E2 -3477.211} C_VEL
LIN {X 0,Y 545.065,Z 616.715,A -85,B 0,C 180,E1 -3479.811,E2 -3479.811} C_VEL
LIN {X 0,Y 545.028,Z 616.718,A -85,B 0,C 180,E1 -3482.841,E2 -3482.841} C_VEL
LIN {X 0,Y 545.086,Z 616.835,A -85,B 0,C 180,E1 -3483.691,E2 -3483.691} C_VEL
LIN {X 0,Y 545.866,Z 622.036,A -85,B 0,C 180,E1 -3484.604,E2 -3484.604} C_VEL
LIN {X 0,Y 545.54,Z 638.911,A -85,B 0,C 180,E1 -3487.406,E2 -3487.406} C_VEL
LIN {X 0,Y 547.432,Z 649.176,A -85,B 0,C 180,E1 -3487.612,E2 -3487.612} C_VEL
LIN {X 0,Y 546.933,Z 775.309,A -85,B 0,C 180,E1 -3489.306,E2 -3489.306} C_VEL
LIN {X 0,Y 546.733,Z 789.476,A -85,B 0,C 180,E1 -3489.643,E2 -3489.643} C_VEL
LIN {X 0,Y 546.562,Z 802.437,A -85,B 0,C 180,E1 -3490.09,E2 -3490.09} C_VEL
LIN {X 0,Y 546.294,Z 814.9,A -85,B 0,C 180,E1 -3490.654,E2 -3490.654} C_VEL
LIN {X 0,Y 546.022,Z 826.687,A -85,B 0,C 180,E1 -3491.327,E2 -3491.327} C_VEL
LIN {X 0,Y 545.746,Z 838.072,A -85,B 0,C 180,E1 -3492.124,E2 -3492.124} C_VEL
LIN {X 0,Y 545.47,Z 849.988,A -85,B 0,C 180,E1 -3493.148,E2 -3493.148} C_VEL
LIN {X 0,Y 545.207,Z 860.895,A -85,B 0,C 180,E1 -3494.294,E2 -3494.294} C_VEL
LIN {X 0,Y 545.009,Z 870.57,A -85,B 0,C 180,E1 -3495.535,E2 -3495.535} C_VEL
LIN {X 0,Y 544.824,Z 878.412,A -85,B 0,C 180,E1 -3496.764,E2 -3496.764} C_VEL
LIN {X 0,Y 544.733,Z 885.258,A -85,B 0,C 180,E1 -3498.087,E2 -3498.087} C_VEL
LIN {X 0,Y 544.692,Z 889.939,A -85,B 0,C 180,E1 -3499.217,E2 -3499.217} C_VEL
LIN {X 0,Y 544.619,Z 894.769,A -85,B 0,C 180,E1 -3500.717,E2 -3500.717} C_VEL
LIN {X 0,Y 544.619,Z 897.355,A -85,B 0,C 180,E1 -3501.839,E2 -3501.839} C_VEL
LIN {X 0,Y 544.652,Z 899.586,A -85,B 0,C 180,E1 -3503.331,E2 -3503.331} C_VEL
LIN {X 0,Y 544.597,Z 900.458,A -85,B 0,C 180,E1 -3504.817,E2 -3504.817} C_VEL
LIN {X 0,Y 544.627,Z 900.003,A -85,B 0,C 180,E1 -3506.301,E2 -3506.301} C_VEL
LIN {X 0,Y 544.569,Z 898.221,A -85,B 0,C 180,E1 -3507.781,E2 -3507.781} C_VEL
LIN {X 0,Y 544.552,Z 895.074,A -85,B 0,C 180,E1 -3509.261,E2 -3509.261} C_VEL
LIN {X 0,Y 544.608,Z 890.453,A -85,B 0,C 180,E1 -3510.739,E2 -3510.739} C_VEL
LIN {X 0,Y 544.683,Z 884.22,A -85,B 0,C 180,E1 -3512.218,E2 -3512.218} C_VEL
LIN {X 0,Y 544.875,Z 877.293,A -85,B 0,C 180,E1 -3513.513,E2 -3513.513} C_VEL
LIN {X 0,Y 545.086,Z 868.738,A -85,B 0,C 180,E1 -3514.808,E2 -3514.808} C_VEL
LIN {X 0,Y 545.274,Z 859.823,A -85,B 0,C 180,E1 -3515.918,E2 -3515.918} C_VEL
LIN {X 0,Y 545.485,Z 848.636,A -85,B 0,C 180,E1 -3517.072,E2 -3517.072} C_VEL
LIN {X 0,Y 545.815,Z 836.956,A -85,B 0,C 180,E1 -3518.05,E2 -3518.05} C_VEL
LIN {X 0,Y 546.08,Z 824.711,A -85,B 0,C 180,E1 -3518.884,E2 -3518.884} C_VEL
LIN {X 0,Y 546.339,Z 812.95,A -85,B 0,C 180,E1 -3519.533,E2 -3519.533} C_VEL
LIN {X 0,Y 546.576,Z 800.149,A -85,B 0,C 180,E1 -3520.09,E2 -3520.09} C_VEL
LIN {X 0,Y 546.766,Z 786.465,A -85,B 0,C 180,E1 -3520.531,E2 -3520.531} C_VEL
LIN {X 0,Y 546.933,Z 772.349,A -85,B 0,C 180,E1 -3520.832,E2 -3520.832} C_VEL
LIN {X 0,Y 547.345,Z 647.884,A -85,B 0,C 180,E1 -3522.499,E2 -3522.499} C_VEL
LIN {X 0,Y 545.588,Z 638.825,A -85,B 0,C 180,E1 -3522.697,E2 -3522.697} C_VEL
LIN {X 0,Y 545.904,Z 622.093,A -85,B 0,C 180,E1 -3525.475,E2 -3525.475} C_VEL
LIN {X 0,Y 545.079,Z 616.717,A -85,B 0,C 180,E1 -3526.431,E2 -3526.431} C_VEL
LIN {X 0,Y 545.095,Z 616.708,A -85,B 0,C 180,E1 -3529.744,E2 -3529.744} C_VEL
LIN {X 0,Y 545.032,Z 616.722,A -85,B 0,C 180,E1 -3532.758,E2 -3532.758} C_VEL
LIN {X 0,Y 545.01,Z 616.717,A -85,B 0,C 180,E1 -3535.489,E2 -3535.489} C_VEL
LIN {X 0,Y 545.002,Z 616.718,A -85,B 0,C 180,E1 -3537.661,E2 -3537.661} C_VEL
LIN {X 0,Y 545.027,Z 616.716,A -85,B 0,C 180,E1 -3540.236,E2 -3540.236} C_VEL
LIN {X 0,Y 545.062,Z 616.716,A -85,B 0,C 180,E1 -3543.059,E2 -3543.059} C_VEL
LIN {X 0,Y 545.021,Z 616.715,A -85,B 0,C 180,E1 -3545.67,E2 -3545.67} C_VEL
LIN {X 0,Y 545.046,Z 616.712,A -85,B 0,C 180,E1 -3548.238,E2 -3548.238} C_VEL
LIN {X 0,Y 545.017,Z 616.722,A -85,B 0,C 180,E1 -3551.121,E2 -3551.121} C_VEL
LIN {X 0,Y 545.034,Z 616.711,A -85,B 0,C 180,E1 -3554.132,E2 -3554.132} C_VEL
LIN {X 0,Y 545.02,Z 616.721,A -85,B 0,C 180,E1 -3556.887,E2 -3556.887} C_VEL
LIN {X 0,Y 545.057,Z 616.71,A -85,B 0,C 180,E1 -3559.856,E2 -3559.856} C_VEL
LIN {X 0,Y 545.027,Z 616.711,A -85,B 0,C 180,E1 -3562.695,E2 -3562.695} C_VEL
LIN {X 0,Y 545.058,Z 616.713,A -85,B 0,C 180,E1 -3565.611,E2 -3565.611} C_VEL
LIN {X 0,Y 545.061,Z 616.708,A -85,B 0,C 180,E1 -3568.321,E2 -3568.321} C_VEL
LIN {X 0,Y 545.067,Z 616.715,A -85,B 0,C 180,E1 -3571.257,E2 -3571.257} C_VEL
LIN {X 0,Y 545.041,Z 616.712,A -85,B 0,C 180,E1 -3573.997,E2 -3573.997} C_VEL
LIN {X 0,Y 545.077,Z 616.704,A -85,B 0,C 180,E1 -3576.44,E2 -3576.44} C_VEL
LIN {X 0,Y 545.095,Z 616.711,A -85,B 0,C 180,E1 -3579.628,E2 -3579.628} C_VEL
LIN {X 0,Y 545.074,Z 616.704,A -85,B 0,C 180,E1 -3582.749,E2 -3582.749} C_VEL
LIN {X 0,Y 545.096,Z 616.71,A -85,B 0,C 180,E1 -3585.82,E2 -3585.82} C_VEL
LIN {X 0,Y 545.121,Z 616.7,A -85,B 0,C 180,E1 -3588.849,E2 -3588.849} C_VEL
LIN {X 0,Y 545.127,Z 616.708,A -85,B 0,C 180,E1 -3591.847,E2 -3591.847} C_VEL
LIN {X 0,Y 545.197,Z 616.692,A -85,B 0,C 180,E1 -3594.823,E2 -3594.823} C_VEL
LIN {X 0,Y 545.197,Z 616.702,A -85,B 0,C 180,E1 -3597.783,E2 -3597.783} C_VEL
LIN {X 0,Y 545.213,Z 616.688,A -85,B 0,C 180,E1 -3600.738,E2 -3600.738} C_VEL
LIN {X 0,Y 545.172,Z 616.695,A -85,B 0,C 180,E1 -3602.956,E2 -3602.956} C_VEL
LIN {X 0,Y 545.167,Z 616.704,A -85,B 0,C 180,E1 -3605.919,E2 -3605.919} C_VEL
LIN {X 0,Y 545.113,Z 616.702,A -85,B 0,C 180,E1 -3608.9,E2 -3608.9} C_VEL
LIN {X 0,Y 545.138,Z 616.706,A -85,B 0,C 180,E1 -3611.904,E2 -3611.904} C_VEL
LIN {X 0,Y 545.089,Z 616.704,A -85,B 0,C 180,E1 -3614.943,E2 -3614.943} C_VEL
LIN {X 0,Y 545.082,Z 616.715,A -85,B 0,C 180,E1 -3618.026,E2 -3618.026} C_VEL
LIN {X 0,Y 545.099,Z 616.71,A -85,B 0,C 180,E1 -3620.372,E2 -3620.372} C_VEL
LIN {X 0,Y 545.082,Z 616.707,A -85,B 0,C 180,E1 -3623.559,E2 -3623.559} C_VEL
LIN {X 0,Y 545.082,Z 616.712,A -85,B 0,C 180,E1 -3626,E2 -3626} C_VEL
LIN {X 0,Y 545.092,Z 616.708,A -85,B 0,C 180,E1 -3628.748,E2 -3628.748} C_VEL
LIN {X 0,Y 545.062,Z 616.71,A -85,B 0,C 180,E1 -3631.679,E2 -3631.679} C_VEL
LIN {X 0,Y 545.08,Z 616.716,A -85,B 0,C 180,E1 -3634.392,E2 -3634.392} C_VEL
LIN {X 0,Y 545.039,Z 616.712,A -85,B 0,C 180,E1 -3637.304,E2 -3637.304} C_VEL
LIN {X 0,Y 545.095,Z 616.709,A -85,B 0,C 180,E1 -3640.14,E2 -3640.14} C_VEL
LIN {X 0,Y 545.08,Z 616.708,A -85,B 0,C 180,E1 -3643.106,E2 -3643.106} C_VEL
LIN {X 0,Y 545.065,Z 616.713,A -85,B 0,C 180,E1 -3646.225,E2 -3646.225} C_VEL
LIN {X 0,Y 545.1,Z 616.71,A -85,B 0,C 180,E1 -3648.887,E2 -3648.887} C_VEL
LIN {X 0,Y 545.054,Z 616.71,A -85,B 0,C 180,E1 -3651.763,E2 -3651.763} C_VEL
LIN {X 0,Y 545.068,Z 616.716,A -85,B 0,C 180,E1 -3654.534,E2 -3654.534} C_VEL
LIN {X 0,Y 545.084,Z 616.71,A -85,B 0,C 180,E1 -3657.212,E2 -3657.212} C_VEL
LIN {X 0,Y 545.069,Z 616.71,A -85,B 0,C 180,E1 -3659.811,E2 -3659.811} C_VEL
LIN {X 0,Y 545.094,Z 616.71,A -85,B 0,C 180,E1 -3662.344,E2 -3662.344} C_VEL
LIN {X 0,Y 545.137,Z 616.741,A -85,B 0,C 180,E1 -3664.168,E2 -3664.168} C_VEL
LIN {X 0,Y 546.945,Z 625.904,A -85,B 0,C 180,E1 -3665.518,E2 -3665.518} C_VEL
LIN {X 0,Y 546.507,Z 644.918,A -85,B 0,C 180,E1 -3668.103,E2 -3668.103} C_VEL
LIN {X 0,Y 546.108,Z 665.144,A -85,B 0,C 180,E1 -3670.842,E2 -3670.842} C_VEL
LIN {X 0,Y 545.868,Z 676.454,A -85,B 0,C 180,E1 -3672.355,E2 -3672.355} C_VEL
LIN {X 0,Y 547.491,Z 685.614,A -85,B 0,C 180,E1 -3672.534,E2 -3672.534} C_VEL
LIN {X 0,Y 546.905,Z 814.878,A -85,B 0,C 180,E1 -3674.272,E2 -3674.272} C_VEL
LIN {X 0,Y 546.682,Z 829.474,A -85,B 0,C 180,E1 -3674.627,E2 -3674.627} C_VEL
LIN {X 0,Y 546.477,Z 843.834,A -85,B 0,C 180,E1 -3675.143,E2 -3675.143} C_VEL
LIN {X 0,Y 546.261,Z 856.638,A -85,B 0,C 180,E1 -3675.756,E2 -3675.756} C_VEL
LIN {X 0,Y 545.944,Z 869.101,A -85,B 0,C 180,E1 -3676.507,E2 -3676.507} C_VEL
LIN {X 0,Y 545.666,Z 881.643,A -85,B 0,C 180,E1 -3677.447,E2 -3677.447} C_VEL
LIN {X 0,Y 545.433,Z 892.946,A -85,B 0,C 180,E1 -3678.491,E2 -3678.491} C_VEL
LIN {X 0,Y 545.175,Z 902.851,A -85,B 0,C 180,E1 -3679.602,E2 -3679.602} C_VEL
LIN {X 0,Y 544.999,Z 911.173,A -85,B 0,C 180,E1 -3680.724,E2 -3680.724} C_VEL
LIN {X 0,Y 544.833,Z 919.127,A -85,B 0,C 180,E1 -3682.029,E2 -3682.029} C_VEL
LIN {X 0,Y 544.753,Z 925.876,A -85,B 0,C 180,E1 -3683.412,E2 -3683.412} C_VEL
LIN {X 0,Y 544.645,Z 931.201,A -85,B 0,C 180,E1 -3684.818,E2 -3684.818} C_VEL
LIN {X 0,Y 544.658,Z 935.316,A -85,B 0,C 180,E1 -3686.301,E2 -3686.301} C_VEL
LIN {X 0,Y 544.568,Z 938.001,A -85,B 0,C 180,E1 -3687.781,E2 -3687.781} C_VEL
LIN {X 0,Y 544.536,Z 939.333,A -85,B 0,C 180,E1 -3689.26,E2 -3689.26} C_VEL
LIN {X 0,Y 544.536,Z 939.333,A -85,B 0,C 180,E1 -3690.739,E2 -3690.739} C_VEL
LIN {X 0,Y 544.568,Z 938.003,A -85,B 0,C 180,E1 -3692.219,E2 -3692.219} C_VEL
LIN {X 0,Y 544.657,Z 935.319,A -85,B 0,C 180,E1 -3693.699,E2 -3693.699} C_VEL
LIN {X 0,Y 544.645,Z 931.202,A -85,B 0,C 180,E1 -3695.182,E2 -3695.182} C_VEL
LIN {X 0,Y 544.734,Z 925.949,A -85,B 0,C 180,E1 -3696.571,E2 -3696.571} C_VEL
LIN {X 0,Y 544.833,Z 919.128,A -85,B 0,C 180,E1 -3697.971,E2 -3697.971} C_VEL
LIN {X 0,Y 544.999,Z 911.174,A -85,B 0,C 180,E1 -3699.276,E2 -3699.276} C_VEL
LIN {X 0,Y 545.175,Z 902.852,A -85,B 0,C 180,E1 -3700.398,E2 -3700.398} C_VEL
LIN {X 0,Y 545.364,Z 893.028,A -85,B 0,C 180,E1 -3701.501,E2 -3701.501} C_VEL
LIN {X 0,Y 545.666,Z 881.644,A -85,B 0,C 180,E1 -3702.553,E2 -3702.553} C_VEL
LIN {X 0,Y 545.944,Z 869.105,A -85,B 0,C 180,E1 -3703.493,E2 -3703.493} C_VEL
LIN {X 0,Y 546.259,Z 856.642,A -85,B 0,C 180,E1 -3704.244,E2 -3704.244} C_VEL
LIN {X 0,Y 546.52,Z 842.7,A -85,B 0,C 180,E1 -3704.903,E2 -3704.903} C_VEL
LIN {X 0,Y 546.72,Z 828.694,A -85,B 0,C 180,E1 -3705.396,E2 -3705.396} C_VEL
LIN {X 0,Y 546.908,Z 814.883,A -85,B 0,C 180,E1 -3705.728,E2 -3705.728} C_VEL
LIN {X 0,Y 547.384,Z 684.868,A -85,B 0,C 180,E1 -3707.48,E2 -3707.48} C_VEL
LIN {X 0,Y 545.866,Z 676.365,A -85,B 0,C 180,E1 -3707.657,E2 -3707.657} C_VEL
LIN {X 0,Y 546.311,Z 655.032,A -85,B 0,C 180,E1 -3710.521,E2 -3710.521} C_VEL
LIN {X 0,Y 546.796,Z 633.242,A -85,B 0,C 180,E1 -3713.481,E2 -3713.481} C_VEL
LIN {X 0,Y 546.923,Z 625.889,A -85,B 0,C 180,E1 -3714.482,E2 -3714.482} C_VEL
LIN {X 0,Y 545.13,Z 616.707,A -85,B 0,C 180,E1 -3715.865,E2 -3715.865} C_VEL
LIN {X 0,Y 545.092,Z 616.711,A -85,B 0,C 180,E1 -3718.748,E2 -3718.748} C_VEL
LIN {X 0,Y 545.08,Z 616.71,A -85,B 0,C 180,E1 -3721.682,E2 -3721.682} C_VEL
LIN {X 0,Y 545.084,Z 616.706,A -85,B 0,C 180,E1 -3724.563,E2 -3724.563} C_VEL
LIN {X 0,Y 545.07,Z 616.716,A -85,B 0,C 180,E1 -3727.301,E2 -3727.301} C_VEL
LIN {X 0,Y 545.076,Z 616.707,A -85,B 0,C 180,E1 -3730.142,E2 -3730.142} C_VEL
LIN {X 0,Y 545.086,Z 616.711,A -85,B 0,C 180,E1 -3733.106,E2 -3733.106} C_VEL
LIN {X 0,Y 545.068,Z 616.709,A -85,B 0,C 180,E1 -3736.224,E2 -3736.224} C_VEL
LIN {X 0,Y 545.103,Z 616.703,A -85,B 0,C 180,E1 -3738.887,E2 -3738.887} C_VEL
LIN {X 0,Y 545.056,Z 616.713,A -85,B 0,C 180,E1 -3741.763,E2 -3741.763} C_VEL
LIN {X 0,Y 545.067,Z 616.708,A -85,B 0,C 180,E1 -3744.534,E2 -3744.534} C_VEL
LIN {X 0,Y 545.084,Z 616.708,A -85,B 0,C 180,E1 -3747.213,E2 -3747.213} C_VEL
LIN {X 0,Y 545.068,Z 616.714,A -85,B 0,C 180,E1 -3749.811,E2 -3749.811} C_VEL
LIN {X 0,Y 545.096,Z 616.706,A -85,B 0,C 180,E1 -3752.345,E2 -3752.345} C_VEL
LIN {X 0,Y 545.119,Z 616.701,A -85,B 0,C 180,E1 -3754.821,E2 -3754.821} C_VEL
LIN {X 0,Y 545.046,Z 616.711,A -85,B 0,C 180,E1 -3757.243,E2 -3757.243} C_VEL
LIN {X 0,Y 545.123,Z 616.704,A -85,B 0,C 180,E1 -3760.415,E2 -3760.415} C_VEL
LIN {X 0,Y 545.078,Z 616.709,A -85,B 0,C 180,E1 -3763.521,E2 -3763.521} C_VEL
LIN {X 0,Y 545.097,Z 616.71,A -85,B 0,C 180,E1 -3765.82,E2 -3765.82} C_VEL
LIN {X 0,Y 545.121,Z 616.702,A -85,B 0,C 180,E1 -3768.85,E2 -3768.85} C_VEL
LIN {X 0,Y 545.129,Z 616.703,A -85,B 0,C 180,E1 -3771.847,E2 -3771.847} C_VEL
LIN {X 0,Y 545.205,Z 616.691,A -85,B 0,C 180,E1 -3774.823,E2 -3774.823} C_VEL
LIN {X 0,Y 545.197,Z 616.694,A -85,B 0,C 180,E1 -3777.784,E2 -3777.784} C_VEL
LIN {X 0,Y 545.212,Z 616.693,A -85,B 0,C 180,E1 -3780.739,E2 -3780.739} C_VEL
LIN {X 0,Y 545.171,Z 616.697,A -85,B 0,C 180,E1 -3782.956,E2 -3782.956} C_VEL
LIN {X 0,Y 545.173,Z 616.695,A -85,B 0,C 180,E1 -3785.92,E2 -3785.92} C_VEL
LIN {X 0,Y 545.112,Z 616.706,A -85,B 0,C 180,E1 -3788.9,E2 -3788.9} C_VEL
LIN {X 0,Y 545.137,Z 616.7,A -85,B 0,C 180,E1 -3791.904,E2 -3791.904} C_VEL
LIN {X 0,Y 545.088,Z 616.709,A -85,B 0,C 180,E1 -3794.944,E2 -3794.944} C_VEL
LIN {X 0,Y 545.074,Z 616.709,A -85,B 0,C 180,E1 -3798.026,E2 -3798.026} C_VEL
LIN {X 0,Y 545.095,Z 616.708,A -85,B 0,C 180,E1 -3800.372,E2 -3800.372} C_VEL
LIN {X 0,Y 545.08,Z 616.706,A -85,B 0,C 180,E1 -3803.56,E2 -3803.56} C_VEL
LIN {X 0,Y 545.076,Z 616.708,A -85,B 0,C 180,E1 -3806.001,E2 -3806.001} C_VEL
LIN {X 0,Y 545.071,Z 616.712,A -85,B 0,C 180,E1 -3808.744,E2 -3808.744} C_VEL
LIN {X 0,Y 545.06,Z 616.71,A -85,B 0,C 180,E1 -3811.679,E2 -3811.679} C_VEL
LIN {X 0,Y 545.06,Z 616.712,A -85,B 0,C 180,E1 -3814.565,E2 -3814.565} C_VEL
LIN {X 0,Y 545.063,Z 616.717,A -85,B 0,C 180,E1 -3817.006,E2 -3817.006} C_VEL
LIN {X 0,Y 544.356,Z 616.802,A -85,B 0,C 180,E1 -3817.622,E2 -3817.622} C_VEL
LIN {X 0,Y 541.489,Z 617.158,A -85,B 0,C 180,E1 -3818.623,E2 -3818.623} C_VEL
LIN {X 0,Y 539.095,Z 617.455,A -85,B 0,C 180,E1 -3819.429,E2 -3819.429} C_VEL
LIN {X 0,Y 538.073,Z 617.578,A -85,B 0,C 180,E1 -3820.051,E2 -3820.051} C_VEL
LIN {X 0,Y 537.992,Z 617.588,A -85,B 0,C 180,E1 -3820.261,E2 -3820.261} C_VEL
LIN {X 0,Y 537.982,Z 617.598,A -85,B 0,C 180,E1 -3822.982,E2 -3822.982} C_VEL
LIN {X 0,Y 538.013,Z 617.588,A -85,B 0,C 180,E1 -3825.928,E2 -3825.928} C_VEL
LIN {X 0,Y 538.008,Z 617.599,A -85,B 0,C 180,E1 -3829.258,E2 -3829.258} C_VEL
LIN {X 0,Y 537.991,Z 617.591,A -85,B 0,C 180,E1 -3832.122,E2 -3832.122} C_VEL
LIN {X 0,Y 537.992,Z 617.592,A -85,B 0,C 180,E1 -3834.915,E2 -3834.915} C_VEL
LIN {X 0,Y 538.015,Z 617.592,A -85,B 0,C 180,E1 -3837.617,E2 -3837.617} C_VEL
LIN {X 0,Y 538.002,Z 617.591,A -85,B 0,C 180,E1 -3840.238,E2 -3840.238} C_VEL
LIN {X 0,Y 538.027,Z 617.595,A -85,B 0,C 180,E1 -3843.424,E2 -3843.424} C_VEL
LIN {X 0,Y 538.047,Z 617.803,A -85,B 0,C 180,E1 -3843.529,E2 -3843.529} C_VEL
LIN {X 0,Y 538.927,Z 623.211,A -85,B 0,C 180,E1 -3844.511,E2 -3844.511} C_VEL
LIN {X 0,Y 538.596,Z 638.873,A -85,B 0,C 180,E1 -3847.164,E2 -3847.164} C_VEL
LIN {X 0,Y 540.674,Z 649.749,A -85,B 0,C 180,E1 -3847.394,E2 -3847.394} C_VEL
LIN {X 0,Y 540.116,Z 775.57,A -85,B 0,C 180,E1 -3849.108,E2 -3849.108} C_VEL
LIN {X 0,Y 539.885,Z 789.547,A -85,B 0,C 180,E1 -3849.445,E2 -3849.445} C_VEL
LIN {X 0,Y 539.65,Z 803.605,A -85,B 0,C 180,E1 -3849.943,E2 -3849.943} C_VEL
LIN {X 0,Y 539.355,Z 817.248,A -85,B 0,C 180,E1 -3850.593,E2 -3850.593} C_VEL
LIN {X 0,Y 539.024,Z 830.035,A -85,B 0,C 180,E1 -3851.371,E2 -3851.371} C_VEL
LIN {X 0,Y 538.713,Z 841.625,A -85,B 0,C 180,E1 -3852.243,E2 -3852.243} C_VEL
LIN {X 0,Y 538.385,Z 853.253,A -85,B 0,C 180,E1 -3853.311,E2 -3853.311} C_VEL
LIN {X 0,Y 538.136,Z 863.548,A -85,B 0,C 180,E1 -3854.471,E2 -3854.471} C_VEL
LIN {X 0,Y 537.912,Z 872.051,A -85,B 0,C 180,E1 -3855.627,E2 -3855.627} C_VEL
LIN {X 0,Y 537.765,Z 880.142,A -85,B 0,C 180,E1 -3856.971,E2 -3856.971} C_VEL
LIN {X 0,Y 537.627,Z 886.62,A -85,B 0,C 180,E1 -3858.31,E2 -3858.31} C_VEL
LIN {X 0,Y 537.576,Z 891.078,A -85,B 0,C 180,E1 -3859.454,E2 -3859.454} C_VEL
LIN {X 0,Y 537.552,Z 894.583,A -85,B 0,C 180,E1 -3860.594,E2 -3860.594} C_VEL
LIN {X 0,Y 537.518,Z 897.226,A -85,B 0,C 180,E1 -3861.731,E2 -3861.731} C_VEL
LIN {X 0,Y 537.552,Z 899.515,A -85,B 0,C 180,E1 -3863.243,E2 -3863.243} C_VEL
LIN {X 0,Y 537.518,Z 900.444,A -85,B 0,C 180,E1 -3864.749,E2 -3864.749} C_VEL
LIN {X 0,Y 537.545,Z 900.045,A -85,B 0,C 180,E1 -3866.252,E2 -3866.252} C_VEL
LIN {X 0,Y 537.488,Z 898.318,A -85,B 0,C 180,E1 -3867.752,E2 -3867.752} C_VEL
LIN {X 0,Y 537.453,Z 895.232,A -85,B 0,C 180,E1 -3869.251,E2 -3869.251} C_VEL
LIN {X 0,Y 537.513,Z 890.698,A -85,B 0,C 180,E1 -3870.749,E2 -3870.749} C_VEL
LIN {X 0,Y 537.599,Z 884.535,A -85,B 0,C 180,E1 -3872.248,E2 -3872.248} C_VEL
LIN {X 0,Y 537.808,Z 877.681,A -85,B 0,C 180,E1 -3873.559,E2 -3873.559} C_VEL
LIN {X 0,Y 538.027,Z 869.209,A -85,B 0,C 180,E1 -3874.871,E2 -3874.871} C_VEL
LIN {X 0,Y 538.235,Z 860.388,A -85,B 0,C 180,E1 -3875.996,E2 -3875.996} C_VEL
LIN {X 0,Y 538.507,Z 850.598,A -85,B 0,C 180,E1 -3877.038,E2 -3877.038} C_VEL
LIN {X 0,Y 538.816,Z 838.98,A -85,B 0,C 180,E1 -3878.06,E2 -3878.06} C_VEL
LIN {X 0,Y 539.133,Z 827.229,A -85,B 0,C 180,E1 -3878.905,E2 -3878.905} C_VEL
LIN {X 0,Y 539.414,Z 814.283,A -85,B 0,C 180,E1 -3879.657,E2 -3879.657} C_VEL
LIN {X 0,Y 539.716,Z 800.654,A -85,B 0,C 180,E1 -3880.267,E2 -3880.267} C_VEL
LIN {X 0,Y 539.952,Z 786.269,A -85,B 0,C 180,E1 -3880.737,E2 -3880.737} C_VEL
LIN {X 0,Y 540.092,Z 772.05,A -85,B 0,C 180,E1 -3881.042,E2 -3881.042} C_VEL
LIN {X 0,Y 540.572,Z 648.856,A -85,B 0,C 180,E1 -3882.711,E2 -3882.711} C_VEL
LIN {X 0,Y 538.631,Z 638.807,A -85,B 0,C 180,E1 -3882.936,E2 -3882.936} C_VEL
LIN {X 0,Y 538.897,Z 622.65,A -85,B 0,C 180,E1 -3885.681,E2 -3885.681} C_VEL
LIN {X 0,Y 538.019,Z 617.597,A -85,B 0,C 180,E1 -3886.604,E2 -3886.604} C_VEL
LIN {X 0,Y 538.062,Z 617.585,A -85,B 0,C 180,E1 -3889.873,E2 -3889.873} C_VEL
LIN {X 0,Y 538.009,Z 617.593,A -85,B 0,C 180,E1 -3893.072,E2 -3893.072} C_VEL
LIN {X 0,Y 537.972,Z 617.594,A -85,B 0,C 180,E1 -3895.655,E2 -3895.655} C_VEL
LIN {X 0,Y 537.977,Z 617.594,A -85,B 0,C 180,E1 -3898.054,E2 -3898.054} C_VEL
LIN {X 0,Y 537.993,Z 617.598,A -85,B 0,C 180,E1 -3900.629,E2 -3900.629} C_VEL
LIN {X 0,Y 538.002,Z 617.592,A -85,B 0,C 180,E1 -3903.275,E2 -3903.275} C_VEL
LIN {X 0,Y 537.964,Z 617.594,A -85,B 0,C 180,E1 -3906.007,E2 -3906.007} C_VEL
LIN {X 0,Y 538.003,Z 617.597,A -85,B 0,C 180,E1 -3908.832,E2 -3908.832} C_VEL
LIN {X 0,Y 537.984,Z 617.591,A -85,B 0,C 180,E1 -3911.873,E2 -3911.873} C_VEL
LIN {X 0,Y 537.996,Z 617.595,A -85,B 0,C 180,E1 -3914.864,E2 -3914.864} C_VEL
LIN {X 0,Y 537.975,Z 617.6,A -85,B 0,C 180,E1 -3917.209,E2 -3917.209} C_VEL
LIN {X 0,Y 538.003,Z 617.588,A -85,B 0,C 180,E1 -3920.201,E2 -3920.201} C_VEL
LIN {X 0,Y 537.994,Z 617.591,A -85,B 0,C 180,E1 -3923.064,E2 -3923.064} C_VEL
LIN {X 0,Y 538.002,Z 617.59,A -85,B 0,C 180,E1 -3925.825,E2 -3925.825} C_VEL
LIN {X 0,Y 538.011,Z 617.587,A -85,B 0,C 180,E1 -3928.498,E2 -3928.498} C_VEL
LIN {X 0,Y 538.022,Z 617.59,A -85,B 0,C 180,E1 -3931.097,E2 -3931.097} C_VEL
LIN {X 0,Y 537.986,Z 617.595,A -85,B 0,C 180,E1 -3933.63,E2 -3933.63} C_VEL
LIN {X 0,Y 538.01,Z 617.585,A -85,B 0,C 180,E1 -3936.122,E2 -3936.122} C_VEL
LIN {X 0,Y 538.04,Z 617.592,A -85,B 0,C 180,E1 -3939.348,E2 -3939.348} C_VEL
LIN {X 0,Y 538.04,Z 617.579,A -85,B 0,C 180,E1 -3942.468,E2 -3942.468} C_VEL
LIN {X 0,Y 538.066,Z 617.589,A -85,B 0,C 180,E1 -3945.63,E2 -3945.63} C_VEL
LIN {X 0,Y 538.08,Z 617.576,A -85,B 0,C 180,E1 -3948.701,E2 -3948.701} C_VEL
LIN {X 0,Y 538.084,Z 617.587,A -85,B 0,C 180,E1 -3951.739,E2 -3951.739} C_VEL
LIN {X 0,Y 538.152,Z 617.569,A -85,B 0,C 180,E1 -3954.755,E2 -3954.755} C_VEL
LIN {X 0,Y 538.169,Z 617.577,A -85,B 0,C 180,E1 -3957.755,E2 -3957.755} C_VEL
LIN {X 0,Y 538.183,Z 617.564,A -85,B 0,C 180,E1 -3960.748,E2 -3960.748} C_VEL
LIN {X 0,Y 538.138,Z 617.571,A -85,B 0,C 180,E1 -3962.994,E2 -3962.994} C_VEL
LIN {X 0,Y 538.118,Z 617.582,A -85,B 0,C 180,E1 -3965.997,E2 -3965.997} C_VEL
LIN {X 0,Y 538.064,Z 617.581,A -85,B 0,C 180,E1 -3969.018,E2 -3969.018} C_VEL
LIN {X 0,Y 538.086,Z 617.587,A -85,B 0,C 180,E1 -3972.062,E2 -3972.062} C_VEL
LIN {X 0,Y 538.049,Z 617.581,A -85,B 0,C 180,E1 -3975.144,E2 -3975.144} C_VEL
LIN {X 0,Y 538.034,Z 617.59,A -85,B 0,C 180,E1 -3978.27,E2 -3978.27} C_VEL
LIN {X 0,Y 538.043,Z 617.585,A -85,B 0,C 180,E1 -3980.651,E2 -3980.651} C_VEL
LIN {X 0,Y 538.005,Z 617.592,A -85,B 0,C 180,E1 -3983.888,E2 -3983.888} C_VEL
LIN {X 0,Y 538.044,Z 617.589,A -85,B 0,C 180,E1 -3986.366,E2 -3986.366} C_VEL
LIN {X 0,Y 538.033,Z 617.586,A -85,B 0,C 180,E1 -3988.933,E2 -3988.933} C_VEL
LIN {X 0,Y 538.017,Z 617.589,A -85,B 0,C 180,E1 -3991.888,E2 -3991.888} C_VEL
LIN {X 0,Y 538.017,Z 617.593,A -85,B 0,C 180,E1 -3994.618,E2 -3994.618} C_VEL
LIN {X 0,Y 538.007,Z 617.588,A -85,B 0,C 180,E1 -3997.17,E2 -3997.17} C_VEL
LIN {X 0,Y 538.057,Z 617.582,A -85,B 0,C 180,E1 -3999.794,E2 -3999.794} C_VEL
LIN {X 0,Y 538.021,Z 617.591,A -85,B 0,C 180,E1 -4002.786,E2 -4002.786} C_VEL
LIN {X 0,Y 538.034,Z 617.586,A -85,B 0,C 180,E1 -4005.14,E2 -4005.14} C_VEL
LIN {X 0,Y 538.044,Z 617.587,A -85,B 0,C 180,E1 -4008.228,E2 -4008.228} C_VEL
LIN {X 0,Y 538.015,Z 617.59,A -85,B 0,C 180,E1 -4011.169,E2 -4011.169} C_VEL
LIN {X 0,Y 538.032,Z 617.587,A -85,B 0,C 180,E1 -4014.083,E2 -4014.083} C_VEL
LIN {X 0,Y 538.034,Z 617.593,A -85,B 0,C 180,E1 -4016.727,E2 -4016.727} C_VEL
LIN {X 0,Y 538.028,Z 617.588,A -85,B 0,C 180,E1 -4019.556,E2 -4019.556} C_VEL
LIN {X 0,Y 538.048,Z 617.586,A -85,B 0,C 180,E1 -4021.95,E2 -4021.95} C_VEL
LIN {X 0,Y 538.078,Z 617.686,A -85,B 0,C 180,E1 -4023.971,E2 -4023.971} C_VEL
LIN {X 0,Y 540.045,Z 627.131,A -85,B 0,C 180,E1 -4025.39,E2 -4025.39} C_VEL
LIN {X 0,Y 539.59,Z 647.679,A -85,B 0,C 180,E1 -4028.21,E2 -4028.21} C_VEL
LIN {X 0,Y 539.069,Z 669.478,A -85,B 0,C 180,E1 -4031.175,E2 -4031.175} C_VEL
LIN {X 0,Y 538.936,Z 676.379,A -85,B 0,C 180,E1 -4032.111,E2 -4032.111} C_VEL
LIN {X 0,Y 540.725,Z 686.547,A -85,B 0,C 180,E1 -4032.321,E2 -4032.321} C_VEL
LIN {X 0,Y 540.084,Z 814.878,A -85,B 0,C 180,E1 -4034.068,E2 -4034.068} C_VEL
LIN {X 0,Y 539.865,Z 829.428,A -85,B 0,C 180,E1 -4034.427,E2 -4034.427} C_VEL
LIN {X 0,Y 539.613,Z 843.833,A -85,B 0,C 180,E1 -4034.949,E2 -4034.949} C_VEL
LIN {X 0,Y 539.347,Z 856.637,A -85,B 0,C 180,E1 -4035.569,E2 -4035.569} C_VEL
LIN {X 0,Y 538.989,Z 869.099,A -85,B 0,C 180,E1 -4036.33,E2 -4036.33} C_VEL
LIN {X 0,Y 538.704,Z 881.645,A -85,B 0,C 180,E1 -4037.282,E2 -4037.282} C_VEL
LIN {X 0,Y 538.43,Z 891.842,A -85,B 0,C 180,E1 -4038.226,E2 -4038.226} C_VEL
LIN {X 0,Y 538.204,Z 901.332,A -85,B 0,C 180,E1 -4039.276,E2 -4039.276} C_VEL
LIN {X 0,Y 537.968,Z 909.91,A -85,B 0,C 180,E1 -4040.412,E2 -4040.412} C_VEL
LIN {X 0,Y 537.805,Z 918.117,A -85,B 0,C 180,E1 -4041.735,E2 -4041.735} C_VEL
LIN {X 0,Y 537.661,Z 923.863,A -85,B 0,C 180,E1 -4042.867,E2 -4042.867} C_VEL
LIN {X 0,Y 537.654,Z 929.96,A -85,B 0,C 180,E1 -4044.374,E2 -4044.374} C_VEL
LIN {X 0,Y 537.55,Z 933.444,A -85,B 0,C 180,E1 -4045.501,E2 -4045.501} C_VEL
LIN {X 0,Y 537.547,Z 936.832,A -85,B 0,C 180,E1 -4047.002,E2 -4047.002} C_VEL
LIN {X 0,Y 537.446,Z 938.834,A -85,B 0,C 180,E1 -4048.501,E2 -4048.501} C_VEL
LIN {X 0,Y 537.44,Z 939.5,A -85,B 0,C 180,E1 -4050,E2 -4050} C_VEL
LIN {X 0,Y 537.447,Z 938.835,A -85,B 0,C 180,E1 -4051.499,E2 -4051.499} C_VEL
LIN {X 0,Y 537.547,Z 936.835,A -85,B 0,C 180,E1 -4052.998,E2 -4052.998} C_VEL
LIN {X 0,Y 537.55,Z 933.447,A -85,B 0,C 180,E1 -4054.499,E2 -4054.499} C_VEL
LIN {X 0,Y 537.647,Z 928.568,A -85,B 0,C 180,E1 -4056.003,E2 -4056.003} C_VEL
LIN {X 0,Y 537.704,Z 922.054,A -85,B 0,C 180,E1 -4057.51,E2 -4057.51} C_VEL
LIN {X 0,Y 537.86,Z 914.803,A -85,B 0,C 180,E1 -4058.832,E2 -4058.832} C_VEL
LIN {X 0,Y 538.063,Z 905.822,A -85,B 0,C 180,E1 -4060.156,E2 -4060.156} C_VEL
LIN {X 0,Y 538.318,Z 896.393,A -85,B 0,C 180,E1 -4061.293,E2 -4061.293} C_VEL
LIN {X 0,Y 538.567,Z 885.954,A -85,B 0,C 180,E1 -4062.338,E2 -4062.338} C_VEL
LIN {X 0,Y 538.895,Z 874.431,A -85,B 0,C 180,E1 -4063.289,E2 -4063.289} C_VEL
LIN {X 0,Y 539.166,Z 863.222,A -85,B 0,C 180,E1 -4064.05,E2 -4064.05} C_VEL
LIN {X 0,Y 539.48,Z 851.136,A -85,B 0,C 180,E1 -4064.716,E2 -4064.716} C_VEL
LIN {X 0,Y 539.785,Z 839.064,A -85,B 0,C 180,E1 -4065.242,E2 -4065.242} C_VEL
LIN {X 0,Y 539.91,Z 825.455,A -85,B 0,C 180,E1 -4065.688,E2 -4065.688} C_VEL
LIN {X 0,Y 540.126,Z 810.626,A -85,B 0,C 180,E1 -4066.003,E2 -4066.003} C_VEL
LIN {X 0,Y 540.643,Z 685.93,A -85,B 0,C 180,E1 -4067.69,E2 -4067.69} C_VEL
LIN {X 0,Y 538.937,Z 676.377,A -85,B 0,C 180,E1 -4067.89,E2 -4067.89} C_VEL
LIN {X 0,Y 539.464,Z 653.541,A -85,B 0,C 180,E1 -4070.994,E2 -4070.994} C_VEL
LIN {X 0,Y 539.951,Z 631.957,A -85,B 0,C 180,E1 -4073.939,E2 -4073.939} C_VEL
LIN {X 0,Y 539.818,Z 625.621,A -85,B 0,C 180,E1 -4074.826,E2 -4074.826} C_VEL
LIN {X 0,Y 538.068,Z 617.587,A -85,B 0,C 180,E1 -4076.051,E2 -4076.051} C_VEL
LIN {X 0,Y 538.034,Z 617.593,A -85,B 0,C 180,E1 -4078.934,E2 -4078.934} C_VEL
LIN {X 0,Y 538.029,Z 617.586,A -85,B 0,C 180,E1 -4081.89,E2 -4081.89} C_VEL
LIN {X 0,Y 538.034,Z 617.585,A -85,B 0,C 180,E1 -4084.621,E2 -4084.621} C_VEL
LIN {X 0,Y 538.025,Z 617.593,A -85,B 0,C 180,E1 -4087.173,E2 -4087.173} C_VEL
LIN {X 0,Y 538.031,Z 617.587,A -85,B 0,C 180,E1 -4089.796,E2 -4089.796} C_VEL
LIN {X 0,Y 538.024,Z 617.587,A -85,B 0,C 180,E1 -4092.786,E2 -4092.786} C_VEL
LIN {X 0,Y 538.031,Z 617.588,A -85,B 0,C 180,E1 -4095.925,E2 -4095.925} C_VEL
LIN {X 0,Y 538.08,Z 617.582,A -85,B 0,C 180,E1 -4099.249,E2 -4099.249} C_VEL
LIN {X 0,Y 537.996,Z 617.587,A -85,B 0,C 180,E1 -4102.123,E2 -4102.123} C_VEL
LIN {X 0,Y 538.022,Z 617.586,A -85,B 0,C 180,E1 -4104.917,E2 -4104.917} C_VEL
LIN {X 0,Y 538.034,Z 617.59,A -85,B 0,C 180,E1 -4107.618,E2 -4107.618} C_VEL
LIN {X 0,Y 538.02,Z 617.588,A -85,B 0,C 180,E1 -4110.239,E2 -4110.239} C_VEL
LIN {X 0,Y 538.068,Z 617.579,A -85,B 0,C 180,E1 -4112.797,E2 -4112.797} C_VEL
LIN {X 0,Y 538.051,Z 617.583,A -85,B 0,C 180,E1 -4115.293,E2 -4115.293} C_VEL
LIN {X 0,Y 538.018,Z 617.594,A -85,B 0,C 180,E1 -4118.042,E2 -4118.042} C_VEL
LIN {X 0,Y 538.042,Z 617.582,A -85,B 0,C 180,E1 -4120.94,E2 -4120.94} C_VEL
LIN {X 0,Y 538.029,Z 617.585,A -85,B 0,C 180,E1 -4123.299,E2 -4123.299} C_VEL
LIN {X 0,Y 538.066,Z 617.583,A -85,B 0,C 180,E1 -4125.631,E2 -4125.631} C_VEL
LIN {X 0,Y 538.08,Z 617.581,A -85,B 0,C 180,E1 -4128.702,E2 -4128.702} C_VEL
LIN {X 0,Y 538.086,Z 617.579,A -85,B 0,C 180,E1 -4131.74,E2 -4131.74} C_VEL
LIN {X 0,Y 538.163,Z 617.569,A -85,B 0,C 180,E1 -4134.755,E2 -4134.755} C_VEL
LIN {X 0,Y 538.169,Z 617.57,A -85,B 0,C 180,E1 -4137.755,E2 -4137.755} C_VEL
LIN {X 0,Y 538.183,Z 617.568,A -85,B 0,C 180,E1 -4140.748,E2 -4140.748} C_VEL
LIN {X 0,Y 538.138,Z 617.573,A -85,B 0,C 180,E1 -4142.995,E2 -4142.995} C_VEL
LIN {X 0,Y 538.123,Z 617.574,A -85,B 0,C 180,E1 -4145.998,E2 -4145.998} C_VEL
LIN {X 0,Y 538.062,Z 617.582,A -85,B 0,C 180,E1 -4149.018,E2 -4149.018} C_VEL
LIN {X 0,Y 538.085,Z 617.58,A -85,B 0,C 180,E1 -4152.063,E2 -4152.063} C_VEL
LIN {X 0,Y 538.048,Z 617.584,A -85,B 0,C 180,E1 -4155.144,E2 -4155.144} C_VEL
LIN {X 0,Y 538.028,Z 617.589,A -85,B 0,C 180,E1 -4158.271,E2 -4158.271} C_VEL
LIN {X 0,Y 538.04,Z 617.591,A -85,B 0,C 180,E1 -4160.652,E2 -4160.652} C_VEL
LIN {X 0,Y 538.004,Z 617.587,A -85,B 0,C 180,E1 -4163.889,E2 -4163.889} C_VEL
LIN {X 0,Y 538.037,Z 617.587,A -85,B 0,C 180,E1 -4166.367,E2 -4166.367} C_VEL
LIN {X 0,Y 538.032,Z 617.587,A -85,B 0,C 180,E1 -4168.933,E2 -4168.933} C_VEL
LIN {X 0,Y 538.012,Z 617.587,A -85,B 0,C 180,E1 -4171.887,E2 -4171.887} C_VEL
LIN {X 0,Y 538.011,Z 617.59,A -85,B 0,C 180,E1 -4174.617,E2 -4174.617} C_VEL
LIN {X 0,Y 538.006,Z 617.596,A -85,B 0,C 180,E1 -4177.17,E2 -4177.17} C_VEL
LIN {X 0,Y 538.012,Z 617.586,A -85,B 0,C 180,E1 -4179.798,E2 -4179.798} C_VEL
LIN {X 0,Y 537.992,Z 617.588,A -85,B 0,C 180,E1 -4180.261,E2 -4180.261} C_VEL
LIN {X 0,Y 537.33,Z 617.677,A -85,B 0,C 180,E1 -4180.887,E2 -4180.887} C_VEL
LIN {X 0,Y 534.478,Z 618.036,A -85,B 0,C 180,E1 -4181.901,E2 -4181.901} C_VEL
LIN {X 0,Y 532.063,Z 618.338,A -85,B 0,C 180,E1 -4182.718,E2 -4182.718} C_VEL
LIN {X 0,Y 531.024,Z 618.465,A -85,B 0,C 180,E1 -4183.349,E2 -4183.349} C_VEL
LIN {X 0,Y 530.938,Z 618.473,A -85,B 0,C 180,E1 -4183.563,E2 -4183.563} C_VEL
LIN {X 0,Y 530.938,Z 618.47,A -85,B 0,C 180,E1 -4186.503,E2 -4186.503} C_VEL
LIN {X 0,Y 530.953,Z 618.473,A -85,B 0,C 180,E1 -4189.564,E2 -4189.564} C_VEL
LIN {X 0,Y 530.969,Z 618.467,A -85,B 0,C 180,E1 -4192.578,E2 -4192.578} C_VEL
LIN {X 0,Y 530.973,Z 618.473,A -85,B 0,C 180,E1 -4195.309,E2 -4195.309} C_VEL
LIN {X 0,Y 530.961,Z 618.469,A -85,B 0,C 180,E1 -4198.031,E2 -4198.031} C_VEL
LIN {X 0,Y 530.967,Z 618.469,A -85,B 0,C 180,E1 -4200.88,E2 -4200.88} C_VEL
LIN {X 0,Y 531.002,Z 618.61,A -85,B 0,C 180,E1 -4203.334,E2 -4203.334} C_VEL
LIN {X 0,Y 531.961,Z 624.182,A -85,B 0,C 180,E1 -4204.362,E2 -4204.362} C_VEL
LIN {X 0,Y 531.665,Z 639.207,A -85,B 0,C 180,E1 -4206.937,E2 -4206.937} C_VEL
LIN {X 0,Y 533.905,Z 650.961,A -85,B 0,C 180,E1 -4207.18,E2 -4207.18} C_VEL
LIN {X 0,Y 533.288,Z 775.812,A -85,B 0,C 180,E1 -4208.903,E2 -4208.903} C_VEL
LIN {X 0,Y 533.038,Z 790.137,A -85,B 0,C 180,E1 -4209.258,E2 -4209.258} C_VEL
LIN {X 0,Y 532.781,Z 804.296,A -85,B 0,C 180,E1 -4209.774,E2 -4209.774} C_VEL
LIN {X 0,Y 532.446,Z 817.788,A -85,B 0,C 180,E1 -4210.431,E2 -4210.431} C_VEL
LIN {X 0,Y 532.09,Z 830.469,A -85,B 0,C 180,E1 -4211.219,E2 -4211.219} C_VEL
LIN {X 0,Y 531.756,Z 841.97,A -85,B 0,C 180,E1 -4212.101,E2 -4212.101} C_VEL
LIN {X 0,Y 531.42,Z 852.566,A -85,B 0,C 180,E1 -4213.085,E2 -4213.085} C_VEL
LIN {X 0,Y 531.128,Z 863.016,A -85,B 0,C 180,E1 -4214.261,E2 -4214.261} C_VEL
LIN {X 0,Y 530.904,Z 871.611,A -85,B 0,C 180,E1 -4215.433,E2 -4215.433} C_VEL
LIN {X 0,Y 530.699,Z 878.745,A -85,B 0,C 180,E1 -4216.6,E2 -4216.6} C_VEL
LIN {X 0,Y 530.594,Z 884.619,A -85,B 0,C 180,E1 -4217.765,E2 -4217.765} C_VEL
LIN {X 0,Y 530.526,Z 889.592,A -85,B 0,C 180,E1 -4218.968,E2 -4218.968} C_VEL
LIN {X 0,Y 530.462,Z 894.396,A -85,B 0,C 180,E1 -4220.467,E2 -4220.467} C_VEL
LIN {X 0,Y 530.431,Z 897.098,A -85,B 0,C 180,E1 -4221.62,E2 -4221.62} C_VEL
LIN {X 0,Y 530.468,Z 899.445,A -85,B 0,C 180,E1 -4223.152,E2 -4223.152} C_VEL
LIN {X 0,Y 530.441,Z 900.43,A -85,B 0,C 180,E1 -4224.678,E2 -4224.678} C_VEL
LIN {X 0,Y 530.465,Z 900.086,A -85,B 0,C 180,E1 -4226.202,E2 -4226.202} C_VEL
LIN {X 0,Y 530.409,Z 898.415,A -85,B 0,C 180,E1 -4227.722,E2 -4227.722} C_VEL
LIN {X 0,Y 530.355,Z 895.387,A -85,B 0,C 180,E1 -4229.241,E2 -4229.241} C_VEL
LIN {X 0,Y 530.418,Z 890.924,A -85,B 0,C 180,E1 -4230.759,E2 -4230.759} C_VEL
LIN {X 0,Y 530.584,Z 886.502,A -85,B 0,C 180,E1 -4231.898,E2 -4231.898} C_VEL
LIN {X 0,Y 530.708,Z 880.142,A -85,B 0,C 180,E1 -4233.226,E2 -4233.226} C_VEL
LIN {X 0,Y 530.915,Z 872.263,A -85,B 0,C 180,E1 -4234.556,E2 -4234.556} C_VEL
LIN {X 0,Y 531.119,Z 864.047,A -85,B 0,C 180,E1 -4235.696,E2 -4235.696} C_VEL
LIN {X 0,Y 531.358,Z 854.184,A -85,B 0,C 180,E1 -4236.837,E2 -4236.837} C_VEL
LIN {X 0,Y 531.759,Z 843.233,A -85,B 0,C 180,E1 -4237.881,E2 -4237.881} C_VEL
LIN {X 0,Y 532.125,Z 831.023,A -85,B 0,C 180,E1 -4238.832,E2 -4238.832} C_VEL
LIN {X 0,Y 532.367,Z 818.99,A -85,B 0,C 180,E1 -4239.594,E2 -4239.594} C_VEL
LIN {X 0,Y 532.788,Z 805.639,A -85,B 0,C 180,E1 -4240.258,E2 -4240.258} C_VEL
LIN {X 0,Y 533.056,Z 791.716,A -85,B 0,C 180,E1 -4240.781,E2 -4240.781} C_VEL
LIN {X 0,Y 533.222,Z 777.041,A -85,B 0,C 180,E1 -4241.162,E2 -4241.162} C_VEL
LIN {X 0,Y 533.36,Z 751.256,A -85,B 0,C 180,E1 -4241.544,E2 -4241.544} C_VEL
LIN {X 0,Y 533.823,Z 650.008,A -85,B 0,C 180,E1 -4242.926,E2 -4242.926} C_VEL
LIN {X 0,Y 531.675,Z 639.012,A -85,B 0,C 180,E1 -4243.161,E2 -4243.161} C_VEL
LIN {X 0,Y 532.018,Z 624.505,A -85,B 0,C 180,E1 -4245.673,E2 -4245.673} C_VEL
LIN {X 0,Y 530.974,Z 618.474,A -85,B 0,C 180,E1 -4246.806,E2 -4246.806} C_VEL
LIN {X 0,Y 531.018,Z 618.465,A -85,B 0,C 180,E1 -4250.128,E2 -4250.128} C_VEL
LIN {X 0,Y 530.944,Z 618.477,A -85,B 0,C 180,E1 -4252.574,E2 -4252.574} C_VEL
LIN {X 0,Y 530.933,Z 618.475,A -85,B 0,C 180,E1 -4255.061,E2 -4255.061} C_VEL
LIN {X 0,Y 530.954,Z 618.468,A -85,B 0,C 180,E1 -4257.599,E2 -4257.599} C_VEL
LIN {X 0,Y 530.936,Z 618.471,A -85,B 0,C 180,E1 -4260.199,E2 -4260.199} C_VEL
LIN {X 0,Y 530.948,Z 618.477,A -85,B 0,C 180,E1 -4262.868,E2 -4262.868} C_VEL
LIN {X 0,Y 530.934,Z 618.47,A -85,B 0,C 180,E1 -4265.622,E2 -4265.622} C_VEL
LIN {X 0,Y 530.959,Z 618.471,A -85,B 0,C 180,E1 -4268.652,E2 -4268.652} C_VEL
LIN {X 0,Y 530.954,Z 618.47,A -85,B 0,C 180,E1 -4271.44,E2 -4271.44} C_VEL
LIN {X 0,Y 530.967,Z 618.466,A -85,B 0,C 180,E1 -4274.549,E2 -4274.549} C_VEL
LIN {X 0,Y 530.917,Z 618.474,A -85,B 0,C 180,E1 -4277.537,E2 -4277.537} C_VEL
LIN {X 0,Y 530.965,Z 618.466,A -85,B 0,C 180,E1 -4280.554,E2 -4280.554} C_VEL
LIN {X 0,Y 530.938,Z 618.47,A -85,B 0,C 180,E1 -4283.44,E2 -4283.44} C_VEL
LIN {X 0,Y 530.964,Z 618.466,A -85,B 0,C 180,E1 -4286.5,E2 -4286.5} C_VEL
LIN {X 0,Y 530.964,Z 618.471,A -85,B 0,C 180,E1 -4289.357,E2 -4289.357} C_VEL
LIN {X 0,Y 530.963,Z 618.472,A -85,B 0,C 180,E1 -4291.542,E2 -4291.542} C_VEL
LIN {X 0,Y 530.964,Z 618.464,A -85,B 0,C 180,E1 -4294.168,E2 -4294.168} C_VEL
LIN {X 0,Y 530.955,Z 618.463,A -85,B 0,C 180,E1 -4296.603,E2 -4296.603} C_VEL
LIN {X 0,Y 531.002,Z 618.464,A -85,B 0,C 180,E1 -4299.062,E2 -4299.062} C_VEL
LIN {X 0,Y 530.987,Z 618.468,A -85,B 0,C 180,E1 -4301.478,E2 -4301.478} C_VEL
LIN {X 0,Y 530.997,Z 618.46,A -85,B 0,C 180,E1 -4304.65,E2 -4304.65} C_VEL
LIN {X 0,Y 531.031,Z 618.461,A -85,B 0,C 180,E1 -4307.775,E2 -4307.775} C_VEL
LIN {X 0,Y 530.981,Z 618.463,A -85,B 0,C 180,E1 -4310.092,E2 -4310.092} C_VEL
LIN {X 0,Y 531.019,Z 618.459,A -85,B 0,C 180,E1 -4312.394,E2 -4312.394} C_VEL
LIN {X 0,Y 531.11,Z 618.446,A -85,B 0,C 180,E1 -4314.685,E2 -4314.685} C_VEL
LIN {X 0,Y 531.141,Z 618.452,A -85,B 0,C 180,E1 -4317.725,E2 -4317.725} C_VEL
LIN {X 0,Y 531.154,Z 618.439,A -85,B 0,C 180,E1 -4320.758,E2 -4320.758} C_VEL
LIN {X 0,Y 531.105,Z 618.448,A -85,B 0,C 180,E1 -4323.034,E2 -4323.034} C_VEL
LIN {X 0,Y 531.073,Z 618.458,A -85,B 0,C 180,E1 -4326.077,E2 -4326.077} C_VEL
LIN {X 0,Y 531.055,Z 618.457,A -85,B 0,C 180,E1 -4328.37,E2 -4328.37} C_VEL
LIN {X 0,Y 531.055,Z 618.457,A -85,B 0,C 180,E1 -4331.672,E2 -4331.672} C_VEL
LIN {X 0,Y 531.034,Z 618.455,A -85,B 0,C 180,E1 -4334.956,E2 -4334.956} C_VEL
LIN {X 0,Y 531.02,Z 618.462,A -85,B 0,C 180,E1 -4337.722,E2 -4337.722} C_VEL
LIN {X 0,Y 531.003,Z 618.46,A -85,B 0,C 180,E1 -4340.938,E2 -4340.938} C_VEL
LIN {X 0,Y 530.968,Z 618.473,A -85,B 0,C 180,E1 -4344.225,E2 -4344.225} C_VEL
LIN {X 0,Y 531.004,Z 618.461,A -85,B 0,C 180,E1 -4346.744,E2 -4346.744} C_VEL
LIN {X 0,Y 530.984,Z 618.463,A -85,B 0,C 180,E1 -4349.322,E2 -4349.322} C_VEL
LIN {X 0,Y 530.973,Z 618.47,A -85,B 0,C 180,E1 -4352.101,E2 -4352.101} C_VEL
LIN {X 0,Y 530.974,Z 618.467,A -85,B 0,C 180,E1 -4354.851,E2 -4354.851} C_VEL
LIN {X 0,Y 530.968,Z 618.465,A -85,B 0,C 180,E1 -4357.507,E2 -4357.507} C_VEL
LIN {X 0,Y 531.028,Z 618.466,A -85,B 0,C 180,E1 -4360.429,E2 -4360.429} C_VEL
LIN {X 0,Y 530.967,Z 618.465,A -85,B 0,C 180,E1 -4363.494,E2 -4363.494} C_VEL
LIN {X 0,Y 530.967,Z 618.472,A -85,B 0,C 180,E1 -4366.505,E2 -4366.505} C_VEL
LIN {X 0,Y 530.992,Z 618.466,A -85,B 0,C 180,E1 -4368.976,E2 -4368.976} C_VEL
LIN {X 0,Y 530.959,Z 618.467,A -85,B 0,C 180,E1 -4371.529,E2 -4371.529} C_VEL
LIN {X 0,Y 530.985,Z 618.468,A -85,B 0,C 180,E1 -4374.382,E2 -4374.382} C_VEL
LIN {X 0,Y 530.975,Z 618.469,A -85,B 0,C 180,E1 -4377.134,E2 -4377.134} C_VEL
LIN {X 0,Y 530.972,Z 618.467,A -85,B 0,C 180,E1 -4379.803,E2 -4379.803} C_VEL
LIN {X 0,Y 531.019,Z 618.465,A -85,B 0,C 180,E1 -4382.466,E2 -4382.466} C_VEL
LIN {X 0,Y 531.052,Z 618.631,A -85,B 0,C 180,E1 -4383.77,E2 -4383.77} C_VEL
LIN {X 0,Y 533.16,Z 628.705,A -85,B 0,C 180,E1 -4385.308,E2 -4385.308} C_VEL
LIN {X 0,Y 532.661,Z 648.907,A -85,B 0,C 180,E1 -4388.116,E2 -4388.116} C_VEL
LIN {X 0,Y 532.121,Z 672.337,A -85,B 0,C 180,E1 -4391.32,E2 -4391.32} C_VEL
LIN {X 0,Y 532.025,Z 676.436,A -85,B 0,C 180,E1 -4391.878,E2 -4391.878} C_VEL
LIN {X 0,Y 533.979,Z 687.366,A -85,B 0,C 180,E1 -4392.101,E2 -4392.101} C_VEL
LIN {X 0,Y 533.251,Z 814.878,A -85,B 0,C 180,E1 -4393.859,E2 -4393.859} C_VEL
LIN {X 0,Y 533.049,Z 829.21,A -85,B 0,C 180,E1 -4394.215,E2 -4394.215} C_VEL
LIN {X 0,Y 532.798,Z 842.702,A -85,B 0,C 180,E1 -4394.703,E2 -4394.703} C_VEL
LIN {X 0,Y 532.462,Z 856.635,A -85,B 0,C 180,E1 -4395.378,E2 -4395.378} C_VEL
LIN {X 0,Y 532.071,Z 869.097,A -85,B 0,C 180,E1 -4396.148,E2 -4396.148} C_VEL
LIN {X 0,Y 531.721,Z 881.646,A -85,B 0,C 180,E1 -4397.112,E2 -4397.112} C_VEL
LIN {X 0,Y 531.421,Z 892.521,A -85,B 0,C 180,E1 -4398.138,E2 -4398.138} C_VEL
LIN {X 0,Y 531.13,Z 902.852,A -85,B 0,C 180,E1 -4399.324,E2 -4399.324} C_VEL
LIN {X 0,Y 530.928,Z 911.174,A -85,B 0,C 180,E1 -4400.476,E2 -4400.476} C_VEL
LIN {X 0,Y 530.709,Z 919.126,A -85,B 0,C 180,E1 -4401.816,E2 -4401.816} C_VEL
LIN {X 0,Y 530.573,Z 925.527,A -85,B 0,C 180,E1 -4403.153,E2 -4403.153} C_VEL
LIN {X 0,Y 530.513,Z 931.2,A -85,B 0,C 180,E1 -4404.679,E2 -4404.679} C_VEL
LIN {X 0,Y 530.497,Z 935.316,A -85,B 0,C 180,E1 -4406.202,E2 -4406.202} C_VEL
LIN {X 0,Y 530.408,Z 938.002,A -85,B 0,C 180,E1 -4407.722,E2 -4407.722} C_VEL
LIN {X 0,Y 530.339,Z 939.333,A -85,B 0,C 180,E1 -4409.241,E2 -4409.241} C_VEL
LIN {X 0,Y 530.339,Z 939.334,A -85,B 0,C 180,E1 -4410.759,E2 -4410.759} C_VEL
LIN {X 0,Y 530.408,Z 938.004,A -85,B 0,C 180,E1 -4412.278,E2 -4412.278} C_VEL
LIN {X 0,Y 530.497,Z 935.32,A -85,B 0,C 180,E1 -4413.798,E2 -4413.798} C_VEL
LIN {X 0,Y 530.514,Z 931.202,A -85,B 0,C 180,E1 -4415.321,E2 -4415.321} C_VEL
LIN {X 0,Y 530.573,Z 925.527,A -85,B 0,C 180,E1 -4416.847,E2 -4416.847} C_VEL
LIN {X 0,Y 530.709,Z 919.128,A -85,B 0,C 180,E1 -4418.184,E2 -4418.184} C_VEL
LIN {X 0,Y 530.928,Z 911.175,A -85,B 0,C 180,E1 -4419.524,E2 -4419.524} C_VEL
LIN {X 0,Y 531.13,Z 902.853,A -85,B 0,C 180,E1 -4420.676,E2 -4420.676} C_VEL
LIN {X 0,Y 531.454,Z 892.354,A -85,B 0,C 180,E1 -4421.879,E2 -4421.879} C_VEL
LIN {X 0,Y 531.721,Z 881.647,A -85,B 0,C 180,E1 -4422.888,E2 -4422.888} C_VEL
LIN {X 0,Y 532.071,Z 869.102,A -85,B 0,C 180,E1 -4423.852,E2 -4423.852} C_VEL
LIN {X 0,Y 532.461,Z 856.639,A -85,B 0,C 180,E1 -4424.621,E2 -4424.621} C_VEL
LIN {X 0,Y 532.771,Z 843.825,A -85,B 0,C 180,E1 -4425.248,E2 -4425.248} C_VEL
LIN {X 0,Y 533.039,Z 829.344,A -85,B 0,C 180,E1 -4425.78,E2 -4425.78} C_VEL
LIN {X 0,Y 533.267,Z 814.883,A -85,B 0,C 180,E1 -4426.141,E2 -4426.141} C_VEL
LIN {X 0,Y 533.895,Z 686.824,A -85,B 0,C 180,E1 -4427.909,E2 -4427.909} C_VEL
LIN {X 0,Y 532.011,Z 676.383,A -85,B 0,C 180,E1 -4428.13,E2 -4428.13} C_VEL
LIN {X 0,Y 532.547,Z 653.286,A -85,B 0,C 180,E1 -4431.279,E2 -4431.279} C_VEL
LIN {X 0,Y 533.147,Z 630.53,A -85,B 0,C 180,E1 -4434.429,E2 -4434.429} C_VEL
LIN {X 0,Y 532.855,Z 626.851,A -85,B 0,C 180,E1 -4434.965,E2 -4434.965} C_VEL
LIN {X 0,Y 531.015,Z 618.466,A -85,B 0,C 180,E1 -4436.261,E2 -4436.261} C_VEL
LIN {X 0,Y 530.991,Z 618.471,A -85,B 0,C 180,E1 -4439.126,E2 -4439.126} C_VEL
LIN {X 0,Y 530.982,Z 618.463,A -85,B 0,C 180,E1 -4442.103,E2 -4442.103} C_VEL
LIN {X 0,Y 530.991,Z 618.464,A -85,B 0,C 180,E1 -4444.854,E2 -4444.854} C_VEL
LIN {X 0,Y 530.975,Z 618.471,A -85,B 0,C 180,E1 -4447.507,E2 -4447.507} C_VEL
LIN {X 0,Y 530.986,Z 618.461,A -85,B 0,C 180,E1 -4450.432,E2 -4450.432} C_VEL
LIN {X 0,Y 530.97,Z 618.472,A -85,B 0,C 180,E1 -4453.282,E2 -4453.282} C_VEL
LIN {X 0,Y 530.989,Z 618.47,A -85,B 0,C 180,E1 -4455.621,E2 -4455.621} C_VEL
LIN {X 0,Y 531.009,Z 618.458,A -85,B 0,C 180,E1 -4458.566,E2 -4458.566} C_VEL
LIN {X 0,Y 530.97,Z 618.47,A -85,B 0,C 180,E1 -4461.346,E2 -4461.346} C_VEL
LIN {X 0,Y 530.984,Z 618.463,A -85,B 0,C 180,E1 -4464.382,E2 -4464.382} C_VEL
LIN {X 0,Y 530.975,Z 618.465,A -85,B 0,C 180,E1 -4467.134,E2 -4467.134} C_VEL
LIN {X 0,Y 530.972,Z 618.468,A -85,B 0,C 180,E1 -4469.803,E2 -4469.803} C_VEL
LIN {X 0,Y 531.018,Z 618.459,A -85,B 0,C 180,E1 -4472.467,E2 -4472.467} C_VEL
LIN {X 0,Y 531.008,Z 618.459,A -85,B 0,C 180,E1 -4474.943,E2 -4474.943} C_VEL
LIN {X 0,Y 530.974,Z 618.469,A -85,B 0,C 180,E1 -4478.247,E2 -4478.247} C_VEL
LIN {X 0,Y 530.999,Z 618.461,A -85,B 0,C 180,E1 -4480.678,E2 -4480.678} C_VEL
LIN {X 0,Y 530.995,Z 618.461,A -85,B 0,C 180,E1 -4483.071,E2 -4483.071} C_VEL
LIN {X 0,Y 531.021,Z 618.459,A -85,B 0,C 180,E1 -4485.436,E2 -4485.436} C_VEL
LIN {X 0,Y 531.04,Z 618.459,A -85,B 0,C 180,E1 -4488.55,E2 -4488.55} C_VEL
LIN {X 0,Y 531.056,Z 618.453,A -85,B 0,C 180,E1 -4491.63,E2 -4491.63} C_VEL
LIN {X 0,Y 531.122,Z 618.447,A -85,B 0,C 180,E1 -4494.685,E2 -4494.685} C_VEL
LIN {X 0,Y 531.141,Z 618.445,A -85,B 0,C 180,E1 -4497.725,E2 -4497.725} C_VEL
LIN {X 0,Y 531.153,Z 618.444,A -85,B 0,C 180,E1 -4500.758,E2 -4500.758} C_VEL
LIN {X 0,Y 531.105,Z 618.449,A -85,B 0,C 180,E1 -4503.034,E2 -4503.034} C_VEL
LIN {X 0,Y 531.077,Z 618.452,A -85,B 0,C 180,E1 -4506.077,E2 -4506.077} C_VEL
LIN {X 0,Y 531.054,Z 618.462,A -85,B 0,C 180,E1 -4508.371,E2 -4508.371} C_VEL
LIN {X 0,Y 531.054,Z 618.453,A -85,B 0,C 180,E1 -4511.672,E2 -4511.672} C_VEL
LIN {X 0,Y 531.034,Z 618.46,A -85,B 0,C 180,E1 -4514.956,E2 -4514.956} C_VEL
LIN {X 0,Y 530.984,Z 618.463,A -85,B 0,C 180,E1 -4517.724,E2 -4517.724} C_VEL
LIN {X 0,Y 531.027,Z 618.457,A -85,B 0,C 180,E1 -4520.127,E2 -4520.127} C_VEL
LIN {X 0,Y 530.947,Z 618.474,A -85,B 0,C 180,E1 -4522.574,E2 -4522.574} C_VEL
LIN {X 0,Y 531.001,Z 618.467,A -85,B 0,C 180,E1 -4525.058,E2 -4525.058} C_VEL
LIN {X 0,Y 530.972,Z 618.461,A -85,B 0,C 180,E1 -4527.598,E2 -4527.598} C_VEL
LIN {X 0,Y 530.962,Z 618.462,A -85,B 0,C 180,E1 -4530.198,E2 -4530.198} C_VEL
LIN {X 0,Y 530.969,Z 618.474,A -85,B 0,C 180,E1 -4532.867,E2 -4532.867} C_VEL
LIN {X 0,Y 530.956,Z 618.468,A -85,B 0,C 180,E1 -4535.62,E2 -4535.62} C_VEL
LIN {X 0,Y 530.966,Z 618.469,A -85,B 0,C 180,E1 -4538.653,E2 -4538.653} C_VEL
LIN {X 0,Y 530.965,Z 618.47,A -85,B 0,C 180,E1 -4541.439,E2 -4541.439} C_VEL
LIN {X 0,Y 530.938,Z 618.473,A -85,B 0,C 180,E1 -4543.563,E2 -4543.563} C_VEL
LIN {X 0,Y 530.271,Z 618.553,A -85,B 0,C 180,E1 -4544.197,E2 -4544.197} C_VEL
LIN {X 0,Y 527.428,Z 618.912,A -85,B 0,C 180,E1 -4545.226,E2 -4545.226} C_VEL
LIN {X 0,Y 525.018,Z 619.212,A -85,B 0,C 180,E1 -4546.054,E2 -4546.054} C_VEL
LIN {X 0,Y 523.973,Z 619.341,A -85,B 0,C 180,E1 -4546.694,E2 -4546.694} C_VEL
LIN {X 0,Y 523.883,Z 619.351,A -85,B 0,C 180,E1 -4546.91,E2 -4546.91} C_VEL
LIN {X 0,Y 523.915,Z 619.346,A -85,B 0,C 180,E1 -4549.917,E2 -4549.917} C_VEL
LIN {X 0,Y 523.909,Z 619.349,A -85,B 0,C 180,E1 -4552.868,E2 -4552.868} C_VEL
LIN {X 0,Y 523.916,Z 619.348,A -85,B 0,C 180,E1 -4555.709,E2 -4555.709} C_VEL
LIN {X 0,Y 523.914,Z 619.346,A -85,B 0,C 180,E1 -4558.455,E2 -4558.455} C_VEL
LIN {X 0,Y 523.908,Z 619.352,A -85,B 0,C 180,E1 -4561.123,E2 -4561.123} C_VEL
LIN {X 0,Y 523.965,Z 619.477,A -85,B 0,C 180,E1 -4563.137,E2 -4563.137} C_VEL
LIN {X 0,Y 525.083,Z 626.384,A -85,B 0,C 180,E1 -4564.428,E2 -4564.428} C_VEL
LIN {X 0,Y 524.748,Z 639.228,A -85,B 0,C 180,E1 -4566.676,E2 -4566.676} C_VEL
LIN {X 0,Y 527.161,Z 651.811,A -85,B 0,C 180,E1 -4566.951,E2 -4566.951} C_VEL
LIN {X 0,Y 526.514,Z 774.945,A -85,B 0,C 180,E1 -4568.67,E2 -4568.67} C_VEL
LIN {X 0,Y 526.243,Z 789.29,A -85,B 0,C 180,E1 -4569.018,E2 -4569.018} C_VEL
LIN {X 0,Y 525.939,Z 803.506,A -85,B 0,C 180,E1 -4569.533,E2 -4569.533} C_VEL
LIN {X 0,Y 525.587,Z 816.537,A -85,B 0,C 180,E1 -4570.165,E2 -4570.165} C_VEL
LIN {X 0,Y 525.196,Z 829.446,A -85,B 0,C 180,E1 -4570.963,E2 -4570.963} C_VEL
LIN {X 0,Y 524.825,Z 841.405,A -85,B 0,C 180,E1 -4571.88,E2 -4571.88} C_VEL
LIN {X 0,Y 524.45,Z 851.867,A -85,B 0,C 180,E1 -4572.854,E2 -4572.854} C_VEL
LIN {X 0,Y 524.129,Z 862.462,A -85,B 0,C 180,E1 -4574.045,E2 -4574.045} C_VEL
LIN {X 0,Y 523.889,Z 871.159,A -85,B 0,C 180,E1 -4575.233,E2 -4575.233} C_VEL
LIN {X 0,Y 523.634,Z 879.422,A -85,B 0,C 180,E1 -4576.613,E2 -4576.613} C_VEL
LIN {X 0,Y 523.502,Z 886.046,A -85,B 0,C 180,E1 -4577.99,E2 -4577.99} C_VEL
LIN {X 0,Y 523.436,Z 890.621,A -85,B 0,C 180,E1 -4579.166,E2 -4579.166} C_VEL
LIN {X 0,Y 523.378,Z 894.208,A -85,B 0,C 180,E1 -4580.337,E2 -4580.337} C_VEL
LIN {X 0,Y 523.34,Z 896.97,A -85,B 0,C 180,E1 -4581.505,E2 -4581.505} C_VEL
LIN {X 0,Y 523.37,Z 899.374,A -85,B 0,C 180,E1 -4583.059,E2 -4583.059} C_VEL
LIN {X 0,Y 523.345,Z 900.416,A -85,B 0,C 180,E1 -4584.606,E2 -4584.606} C_VEL
LIN {X 0,Y 523.369,Z 900.128,A -85,B 0,C 180,E1 -4586.15,E2 -4586.15} C_VEL
LIN {X 0,Y 523.332,Z 898.512,A -85,B 0,C 180,E1 -4587.691,E2 -4587.691} C_VEL
LIN {X 0,Y 523.26,Z 895.542,A -85,B 0,C 180,E1 -4589.231,E2 -4589.231} C_VEL
LIN {X 0,Y 523.323,Z 891.141,A -85,B 0,C 180,E1 -4590.77,E2 -4590.77} C_VEL
LIN {X 0,Y 523.443,Z 885.164,A -85,B 0,C 180,E1 -4592.309,E2 -4592.309} C_VEL
LIN {X 0,Y 523.69,Z 878.456,A -85,B 0,C 180,E1 -4593.655,E2 -4593.655} C_VEL
LIN {X 0,Y 523.928,Z 870.15,A -85,B 0,C 180,E1 -4595.002,E2 -4595.002} C_VEL
LIN {X 0,Y 524.162,Z 861.52,A -85,B 0,C 180,E1 -4596.158,E2 -4596.158} C_VEL
LIN {X 0,Y 524.516,Z 850.836,A -85,B 0,C 180,E1 -4597.339,E2 -4597.339} C_VEL
LIN {X 0,Y 524.906,Z 839.444,A -85,B 0,C 180,E1 -4598.372,E2 -4598.372} C_VEL
LIN {X 0,Y 525.276,Z 827.791,A -85,B 0,C 180,E1 -4599.239,E2 -4599.239} C_VEL
LIN {X 0,Y 525.578,Z 816.735,A -85,B 0,C 180,E1 -4599.914,E2 -4599.914} C_VEL
LIN {X 0,Y 525.945,Z 803.918,A -85,B 0,C 180,E1 -4600.539,E2 -4600.539} C_VEL
LIN {X 0,Y 526.207,Z 790.165,A -85,B 0,C 180,E1 -4601.045,E2 -4601.045} C_VEL
LIN {X 0,Y 526.43,Z 775.796,A -85,B 0,C 180,E1 -4601.406,E2 -4601.406} C_VEL
LIN {X 0,Y 527.175,Z 651.424,A -85,B 0,C 180,E1 -4603.143,E2 -4603.143} C_VEL
LIN {X 0,Y 524.77,Z 639.147,A -85,B 0,C 180,E1 -4603.426,E2 -4603.426} C_VEL
LIN {X 0,Y 525.111,Z 626.035,A -85,B 0,C 180,E1 -4605.725,E2 -4605.725} C_VEL
LIN {X 0,Y 523.923,Z 619.351,A -85,B 0,C 180,E1 -4607.014,E2 -4607.014} C_VEL
LIN {X 0,Y 523.973,Z 619.343,A -85,B 0,C 180,E1 -4610.131,E2 -4610.131} C_VEL
LIN {X 0,Y 523.91,Z 619.352,A -85,B 0,C 180,E1 -4612.894,E2 -4612.894} C_VEL
LIN {X 0,Y 523.873,Z 619.351,A -85,B 0,C 180,E1 -4615.423,E2 -4615.423} C_VEL
LIN {X 0,Y 523.9,Z 619.348,A -85,B 0,C 180,E1 -4618.003,E2 -4618.003} C_VEL
LIN {X 0,Y 523.902,Z 619.354,A -85,B 0,C 180,E1 -4620.846,E2 -4620.846} C_VEL
LIN {X 0,Y 523.915,Z 619.344,A -85,B 0,C 180,E1 -4623.726,E2 -4623.726} C_VEL
LIN {X 0,Y 523.87,Z 619.352,A -85,B 0,C 180,E1 -4626.396,E2 -4626.396} C_VEL
LIN {X 0,Y 523.906,Z 619.347,A -85,B 0,C 180,E1 -4629.086,E2 -4629.086} C_VEL
LIN {X 0,Y 523.897,Z 619.346,A -85,B 0,C 180,E1 -4632.125,E2 -4632.125} C_VEL
LIN {X 0,Y 523.937,Z 619.346,A -85,B 0,C 180,E1 -4635.311,E2 -4635.311} C_VEL
LIN {X 0,Y 523.917,Z 619.346,A -85,B 0,C 180,E1 -4638.695,E2 -4638.695} C_VEL
LIN {X 0,Y 523.904,Z 619.339,A -85,B 0,C 180,E1 -4641.897,E2 -4641.897} C_VEL
LIN {X 0,Y 523.921,Z 619.344,A -85,B 0,C 180,E1 -4644.912,E2 -4644.912} C_VEL
LIN {X 0,Y 523.938,Z 619.343,A -85,B 0,C 180,E1 -4647.68,E2 -4647.68} C_VEL
LIN {X 0,Y 523.955,Z 619.337,A -85,B 0,C 180,E1 -4650.677,E2 -4650.677} C_VEL
LIN {X 0,Y 523.902,Z 619.348,A -85,B 0,C 180,E1 -4653.724,E2 -4653.724} C_VEL
LIN {X 0,Y 523.912,Z 619.34,A -85,B 0,C 180,E1 -4656.269,E2 -4656.269} C_VEL
LIN {X 0,Y 523.949,Z 619.34,A -85,B 0,C 180,E1 -4658.766,E2 -4658.766} C_VEL
LIN {X 0,Y 523.949,Z 619.344,A -85,B 0,C 180,E1 -4661.22,E2 -4661.22} C_VEL
LIN {X 0,Y 523.93,Z 619.348,A -85,B 0,C 180,E1 -4663.638,E2 -4663.638} C_VEL
LIN {X 0,Y 523.937,Z 619.343,A -85,B 0,C 180,E1 -4666.028,E2 -4666.028} C_VEL
LIN {X 0,Y 523.996,Z 619.333,A -85,B 0,C 180,E1 -4669.177,E2 -4669.177} C_VEL
LIN {X 0,Y 524.001,Z 619.334,A -85,B 0,C 180,E1 -4672.292,E2 -4672.292} C_VEL
LIN {X 0,Y 524.07,Z 619.323,A -85,B 0,C 180,E1 -4674.613,E2 -4674.613} C_VEL
LIN {X 0,Y 524.113,Z 619.326,A -85,B 0,C 180,E1 -4677.694,E2 -4677.694} C_VEL
LIN {X 0,Y 524.124,Z 619.315,A -85,B 0,C 180,E1 -4680.768,E2 -4680.768} C_VEL
LIN {X 0,Y 524.072,Z 619.324,A -85,B 0,C 180,E1 -4683.075,E2 -4683.075} C_VEL
LIN {X 0,Y 524.033,Z 619.333,A -85,B 0,C 180,E1 -4686.159,E2 -4686.159} C_VEL
LIN {X 0,Y 524.003,Z 619.334,A -85,B 0,C 180,E1 -4688.484,E2 -4688.484} C_VEL
LIN {X 0,Y 524.006,Z 619.335,A -85,B 0,C 180,E1 -4691.739,E2 -4691.739} C_VEL
LIN {X 0,Y 523.996,Z 619.331,A -85,B 0,C 180,E1 -4695.052,E2 -4695.052} C_VEL
LIN {X 0,Y 523.967,Z 619.344,A -85,B 0,C 180,E1 -4697.969,E2 -4697.969} C_VEL
LIN {X 0,Y 523.975,Z 619.34,A -85,B 0,C 180,E1 -4700.41,E2 -4700.41} C_VEL
LIN {X 0,Y 523.913,Z 619.343,A -85,B 0,C 180,E1 -4702.893,E2 -4702.893} C_VEL
LIN {X 0,Y 523.987,Z 619.34,A -85,B 0,C 180,E1 -4706.02,E2 -4706.02} C_VEL
LIN {X 0,Y 523.941,Z 619.342,A -85,B 0,C 180,E1 -4708.874,E2 -4708.874} C_VEL
LIN {X 0,Y 523.926,Z 619.342,A -85,B 0,C 180,E1 -4711.544,E2 -4711.544} C_VEL
LIN {X 0,Y 523.937,Z 619.349,A -85,B 0,C 180,E1 -4714.29,E2 -4714.29} C_VEL
LIN {X 0,Y 523.909,Z 619.345,A -85,B 0,C 180,E1 -4717.132,E2 -4717.132} C_VEL
LIN {X 0,Y 523.971,Z 619.34,A -85,B 0,C 180,E1 -4720.134,E2 -4720.134} C_VEL
LIN {X 0,Y 523.923,Z 619.343,A -85,B 0,C 180,E1 -4723.167,E2 -4723.167} C_VEL
LIN {X 0,Y 523.942,Z 619.34,A -85,B 0,C 180,E1 -4725.772,E2 -4725.772} C_VEL
LIN {X 0,Y 523.947,Z 619.345,A -85,B 0,C 180,E1 -4728.908,E2 -4728.908} C_VEL
LIN {X 0,Y 523.92,Z 619.344,A -85,B 0,C 180,E1 -4731.898,E2 -4731.898} C_VEL
LIN {X 0,Y 523.941,Z 619.348,A -85,B 0,C 180,E1 -4734.909,E2 -4734.909} C_VEL
LIN {X 0,Y 523.945,Z 619.341,A -85,B 0,C 180,E1 -4737.678,E2 -4737.678} C_VEL
LIN {X 0,Y 523.957,Z 619.347,A -85,B 0,C 180,E1 -4740.676,E2 -4740.676} C_VEL
LIN {X 0,Y 524,Z 619.44,A -85,B 0,C 180,E1 -4743.542,E2 -4743.542} C_VEL
LIN {X 0,Y 526.287,Z 630.391,A -85,B 0,C 180,E1 -4745.24,E2 -4745.24} C_VEL
LIN {X 0,Y 525.743,Z 650.135,A -85,B 0,C 180,E1 -4748.019,E2 -4748.019} C_VEL
LIN {X 0,Y 525.148,Z 673.559,A -85,B 0,C 180,E1 -4751.265,E2 -4751.265} C_VEL
LIN {X 0,Y 525.08,Z 676.162,A -85,B 0,C 180,E1 -4751.623,E2 -4751.623} C_VEL
LIN {X 0,Y 527.214,Z 688.868,A -85,B 0,C 180,E1 -4751.887,E2 -4751.887} C_VEL
LIN {X 0,Y 526.435,Z 814.872,A -85,B 0,C 180,E1 -4753.644,E2 -4753.644} C_VEL
LIN {X 0,Y 526.236,Z 829.056,A -85,B 0,C 180,E1 -4754.001,E2 -4754.001} C_VEL
LIN {X 0,Y 525.957,Z 842.701,A -85,B 0,C 180,E1 -4754.499,E2 -4754.499} C_VEL
LIN {X 0,Y 525.64,Z 854.869,A -85,B 0,C 180,E1 -4755.085,E2 -4755.085} C_VEL
LIN {X 0,Y 525.198,Z 867.67,A -85,B 0,C 180,E1 -4755.864,E2 -4755.864} C_VEL
LIN {X 0,Y 524.829,Z 879.305,A -85,B 0,C 180,E1 -4756.743,E2 -4756.743} C_VEL
LIN {X 0,Y 524.503,Z 890.07,A -85,B 0,C 180,E1 -4757.73,E2 -4757.73} C_VEL
LIN {X 0,Y 524.241,Z 899.705,A -85,B 0,C 180,E1 -4758.791,E2 -4758.791} C_VEL
LIN {X 0,Y 523.904,Z 908.555,A -85,B 0,C 180,E1 -4759.957,E2 -4759.957} C_VEL
LIN {X 0,Y 523.695,Z 917.033,A -85,B 0,C 180,E1 -4761.316,E2 -4761.316} C_VEL
LIN {X 0,Y 523.507,Z 923.863,A -85,B 0,C 180,E1 -4762.673,E2 -4762.673} C_VEL
LIN {X 0,Y 523.473,Z 928.568,A -85,B 0,C 180,E1 -4763.834,E2 -4763.834} C_VEL
LIN {X 0,Y 523.376,Z 932.38,A -85,B 0,C 180,E1 -4764.993,E2 -4764.993} C_VEL
LIN {X 0,Y 523.419,Z 935.316,A -85,B 0,C 180,E1 -4766.15,E2 -4766.15} C_VEL
LIN {X 0,Y 523.332,Z 938.002,A -85,B 0,C 180,E1 -4767.691,E2 -4767.691} C_VEL
LIN {X 0,Y 523.245,Z 939.334,A -85,B 0,C 180,E1 -4769.23,E2 -4769.23} C_VEL
LIN {X 0,Y 523.245,Z 939.334,A -85,B 0,C 180,E1 -4770.77,E2 -4770.77} C_VEL
LIN {X 0,Y 523.332,Z 938.005,A -85,B 0,C 180,E1 -4772.309,E2 -4772.309} C_VEL
LIN {X 0,Y 523.419,Z 935.32,A -85,B 0,C 180,E1 -4773.849,E2 -4773.849} C_VEL
LIN {X 0,Y 523.452,Z 931.202,A -85,B 0,C 180,E1 -4775.393,E2 -4775.393} C_VEL
LIN {X 0,Y 523.494,Z 925.526,A -85,B 0,C 180,E1 -4776.94,E2 -4776.94} C_VEL
LIN {X 0,Y 523.664,Z 919.127,A -85,B 0,C 180,E1 -4778.295,E2 -4778.295} C_VEL
LIN {X 0,Y 523.863,Z 911.174,A -85,B 0,C 180,E1 -4779.654,E2 -4779.654} C_VEL
LIN {X 0,Y 524.117,Z 902.852,A -85,B 0,C 180,E1 -4780.82,E2 -4780.82} C_VEL
LIN {X 0,Y 524.447,Z 892.089,A -85,B 0,C 180,E1 -4782.068,E2 -4782.068} C_VEL
LIN {X 0,Y 524.779,Z 881.648,A -85,B 0,C 180,E1 -4783.061,E2 -4783.061} C_VEL
LIN {X 0,Y 525.173,Z 869.1,A -85,B 0,C 180,E1 -4784.037,E2 -4784.037} C_VEL
LIN {X 0,Y 525.59,Z 856.638,A -85,B 0,C 180,E1 -4784.817,E2 -4784.817} C_VEL
LIN {X 0,Y 525.93,Z 843.823,A -85,B 0,C 180,E1 -4785.452,E2 -4785.452} C_VEL
LIN {X 0,Y 526.214,Z 830.124,A -85,B 0,C 180,E1 -4785.965,E2 -4785.965} C_VEL
LIN {X 0,Y 526.449,Z 816.019,A -85,B 0,C 180,E1 -4786.331,E2 -4786.331} C_VEL
LIN {X 0,Y 526.624,Z 787.897,A -85,B 0,C 180,E1 -4786.749,E2 -4786.749} C_VEL
LIN {X 0,Y 527.134,Z 687.721,A -85,B 0,C 180,E1 -4788.132,E2 -4788.132} C_VEL
LIN {X 0,Y 525.081,Z 676.16,A -85,B 0,C 180,E1 -4788.376,E2 -4788.376} C_VEL
LIN {X 0,Y 525.639,Z 653.032,A -85,B 0,C 180,E1 -4791.573,E2 -4791.573} C_VEL
LIN {X 0,Y 526.286,Z 631.335,A -85,B 0,C 180,E1 -4794.62,E2 -4794.62} C_VEL
LIN {X 0,Y 525.265,Z 625.253,A -85,B 0,C 180,E1 -4795.545,E2 -4795.545} C_VEL
LIN {X 0,Y 524.005,Z 619.34,A -85,B 0,C 180,E1 -4796.484,E2 -4796.484} C_VEL
LIN {X 0,Y 523.956,Z 619.347,A -85,B 0,C 180,E1 -4799.324,E2 -4799.324} C_VEL
LIN {X 0,Y 523.941,Z 619.34,A -85,B 0,C 180,E1 -4802.449,E2 -4802.449} C_VEL
LIN {X 0,Y 523.938,Z 619.345,A -85,B 0,C 180,E1 -4805.225,E2 -4805.225} C_VEL
LIN {X 0,Y 523.92,Z 619.343,A -85,B 0,C 180,E1 -4808.101,E2 -4808.101} C_VEL
LIN {X 0,Y 523.963,Z 619.343,A -85,B 0,C 180,E1 -4811.311,E2 -4811.311} C_VEL
LIN {X 0,Y 523.957,Z 619.337,A -85,B 0,C 180,E1 -4814.691,E2 -4814.691} C_VEL
LIN {X 0,Y 523.958,Z 619.34,A -85,B 0,C 180,E1 -4817.882,E2 -4817.882} C_VEL
LIN {X 0,Y 523.98,Z 619.34,A -85,B 0,C 180,E1 -4819.923,E2 -4819.923} C_VEL
LIN {X 0,Y 523.913,Z 619.339,A -85,B 0,C 180,E1 -4822.868,E2 -4822.868} C_VEL
LIN {X 0,Y 523.946,Z 619.348,A -85,B 0,C 180,E1 -4825.711,E2 -4825.711} C_VEL
LIN {X 0,Y 523.933,Z 619.334,A -85,B 0,C 180,E1 -4828.457,E2 -4828.457} C_VEL
LIN {X 0,Y 523.942,Z 619.34,A -85,B 0,C 180,E1 -4831.126,E2 -4831.126} C_VEL
LIN {X 0,Y 523.986,Z 619.342,A -85,B 0,C 180,E1 -4833.98,E2 -4833.98} C_VEL
LIN {X 0,Y 523.938,Z 619.343,A -85,B 0,C 180,E1 -4836.271,E2 -4836.271} C_VEL
LIN {X 0,Y 523.948,Z 619.339,A -85,B 0,C 180,E1 -4838.767,E2 -4838.767} C_VEL
LIN {X 0,Y 523.956,Z 619.338,A -85,B 0,C 180,E1 -4841.221,E2 -4841.221} C_VEL
LIN {X 0,Y 523.942,Z 619.343,A -85,B 0,C 180,E1 -4843.639,E2 -4843.639} C_VEL
LIN {X 0,Y 523.942,Z 619.347,A -85,B 0,C 180,E1 -4846.028,E2 -4846.028} C_VEL
LIN {X 0,Y 524.014,Z 619.336,A -85,B 0,C 180,E1 -4848.394,E2 -4848.394} C_VEL
LIN {X 0,Y 524.005,Z 619.331,A -85,B 0,C 180,E1 -4851.516,E2 -4851.516} C_VEL
LIN {X 0,Y 524.083,Z 619.324,A -85,B 0,C 180,E1 -4854.614,E2 -4854.614} C_VEL
LIN {X 0,Y 524.113,Z 619.32,A -85,B 0,C 180,E1 -4857.695,E2 -4857.695} C_VEL
LIN {X 0,Y 524.123,Z 619.319,A -85,B 0,C 180,E1 -4860.769,E2 -4860.769} C_VEL
LIN {X 0,Y 524.071,Z 619.325,A -85,B 0,C 180,E1 -4863.075,E2 -4863.075} C_VEL
LIN {X 0,Y 524.039,Z 619.33,A -85,B 0,C 180,E1 -4866.159,E2 -4866.159} C_VEL
LIN {X 0,Y 524.002,Z 619.342,A -85,B 0,C 180,E1 -4868.484,E2 -4868.484} C_VEL
LIN {X 0,Y 524.006,Z 619.332,A -85,B 0,C 180,E1 -4871.74,E2 -4871.74} C_VEL
LIN {X 0,Y 523.997,Z 619.335,A -85,B 0,C 180,E1 -4875.053,E2 -4875.053} C_VEL
